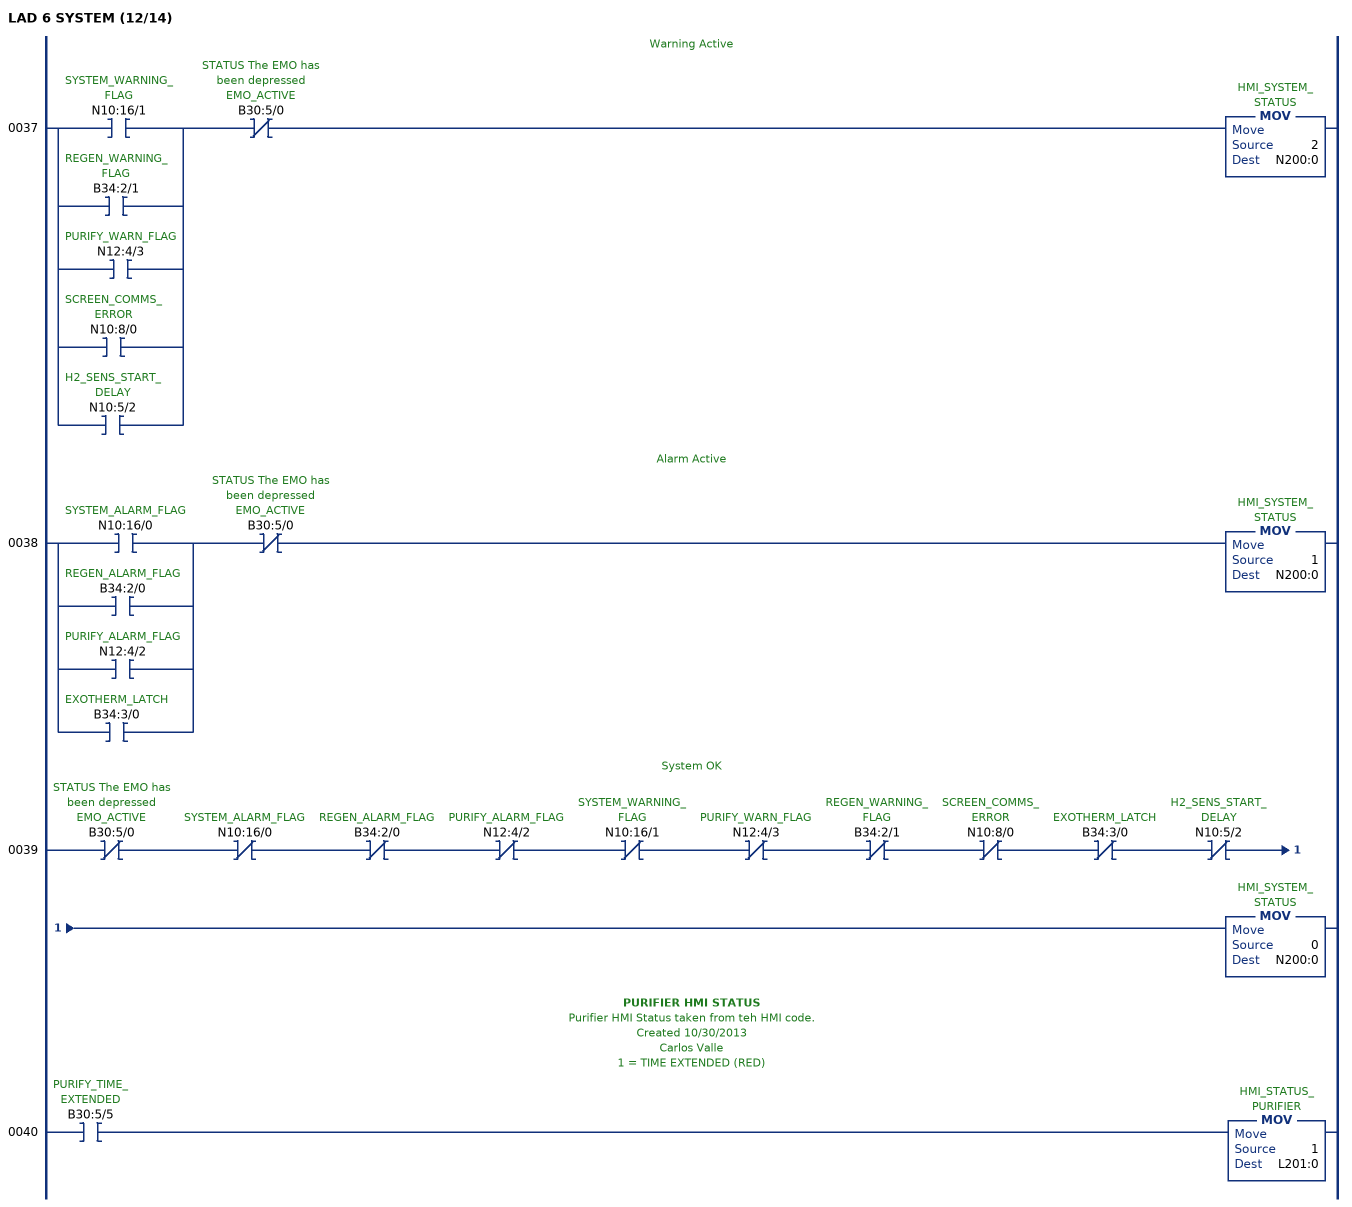
% Rung: 37 %
% Warning Active %
SOR BST XIC N10:16/1 NXB XIC B34:2/1 NXB XIC N12:4/3 NXB XIC N10:8/0 NXB XIC N10:5/2 BND XIO B30:5/0 MOV 2 N200:0 EOR
%   N10:16/1  SYSTEM_WARNING_FLAG %
%   B34:2/1  REGEN_WARNING_FLAG %
%   N12:4/3  PURIFY_WARN_FLAG %
%   N10:8/0  SCREEN_COMMS_ERROR %
%   N10:5/2  H2_SENS_START_DELAY %
%   B30:5/0  EMO_ACTIVE  "STATUS The EMO has been depressed" %
%   N200:0  HMI_SYSTEM_STATUS %
% Rung: 38 %
% Alarm Active %
SOR BST XIC N10:16/0 NXB XIC B34:2/0 NXB XIC N12:4/2 NXB XIC B34:3/0 BND XIO B30:5/0 MOV 1 N200:0 EOR
%   N10:16/0  SYSTEM_ALARM_FLAG %
%   B34:2/0  REGEN_ALARM_FLAG %
%   N12:4/2  PURIFY_ALARM_FLAG %
%   B34:3/0  EXOTHERM_LATCH %
%   B30:5/0  EMO_ACTIVE  "STATUS The EMO has been depressed" %
%   N200:0  HMI_SYSTEM_STATUS %
% Rung: 39 %
% System OK %
SOR XIO B30:5/0 XIO N10:16/0 XIO B34:2/0 XIO N12:4/2 XIO N10:16/1 XIO N12:4/3 XIO B34:2/1 XIO N10:8/0 XIO B34:3/0 XIO N10:5/2 MOV 0 N200:0 EOR
%   B30:5/0  EMO_ACTIVE  "STATUS The EMO has been depressed" %
%   N10:16/0  SYSTEM_ALARM_FLAG %
%   B34:2/0  REGEN_ALARM_FLAG %
%   N12:4/2  PURIFY_ALARM_FLAG %
%   N10:16/1  SYSTEM_WARNING_FLAG %
%   N12:4/3  PURIFY_WARN_FLAG %
%   B34:2/1  REGEN_WARNING_FLAG %
%   N10:8/0  SCREEN_COMMS_ERROR %
%   B34:3/0  EXOTHERM_LATCH %
%   N10:5/2  H2_SENS_START_DELAY %
%   N200:0  HMI_SYSTEM_STATUS %
% Rung: 40 %
% TITLE: PURIFIER HMI STATUS %
% Purifier HMI Status taken from teh HMI code.
% Created 10/30/2013
% Carlos Valle
% 1 = TIME EXTENDED (RED) %
SOR XIC B30:5/5 MOV 1 L201:0 EOR
%   B30:5/5  PURIFY_TIME_EXTENDED %
%   L201:0  HMI_STATUS_PURIFIER %

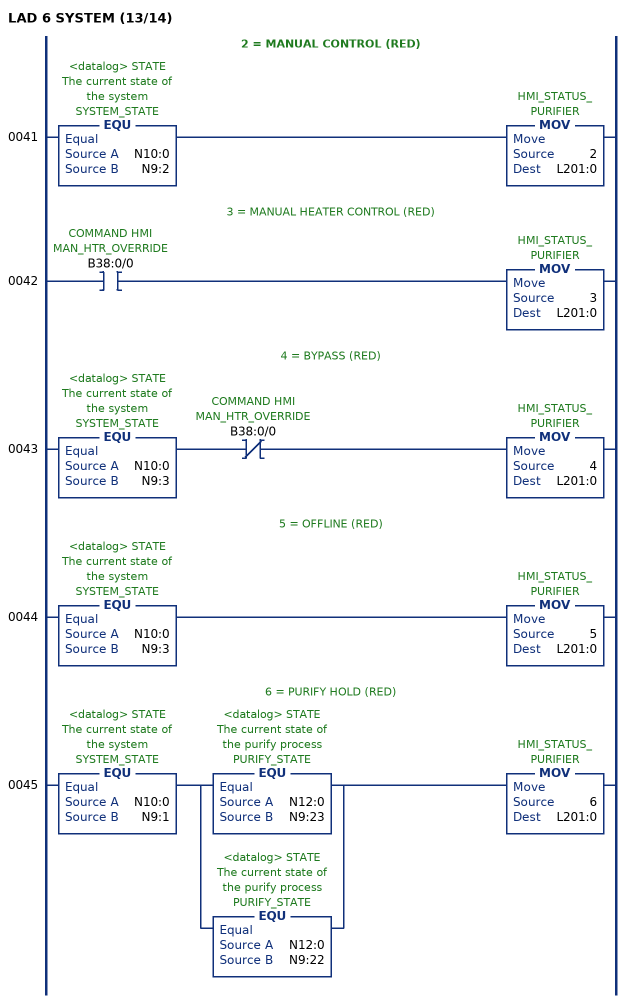
% Rung: 41 %
% TITLE: 2 = MANUAL CONTROL (RED) %
SOR EQU N10:0 N9:2 MOV 2 L201:0 EOR
%   N10:0  SYSTEM_STATE  "<datalog> STATE The current state of the system" %
%   N9:2  SYSTEM_MANUAL  "STATE System Manual" %
%   L201:0  HMI_STATUS_PURIFIER %
% Rung: 42 %
% 3 = MANUAL HEATER CONTROL (RED) %
SOR XIC B38:0/0 MOV 3 L201:0 EOR
%   B38:0/0  MAN_HTR_OVERRIDE  "COMMAND HMI" %
%   L201:0  HMI_STATUS_PURIFIER %
% Rung: 43 %
% 4 = BYPASS (RED) %
SOR EQU N10:0 N9:3 XIO B38:0/0 MOV 4 L201:0 EOR
%   N10:0  SYSTEM_STATE  "<datalog> STATE The current state of the system" %
%   N9:3  SYSTEM_ALARM  "STATE System Alarm" %
%   B38:0/0  MAN_HTR_OVERRIDE  "COMMAND HMI" %
%   L201:0  HMI_STATUS_PURIFIER %
% Rung: 44 %
% 5 = OFFLINE (RED) %
SOR EQU N10:0 N9:3 MOV 5 L201:0 EOR
%   N10:0  SYSTEM_STATE  "<datalog> STATE The current state of the system" %
%   N9:3  SYSTEM_ALARM  "STATE System Alarm" %
%   L201:0  HMI_STATUS_PURIFIER %
% Rung: 45 %
% 6 = PURIFY HOLD (RED) %
SOR EQU N10:0 N9:1 BST EQU N12:0 N9:23 NXB EQU N12:0 N9:22 BND MOV 6 L201:0 EOR
%   N10:0  SYSTEM_STATE  "<datalog> STATE The current state of the system" %
%   N9:1  SYSTEM_PROCESS  "STATE System Process" %
%   N12:0  PURIFY_STATE  "<datalog> STATE The current state of the purify process" %
%   N9:23  PURIFY_MANUAL_HOLD  "STATE Purify Manual Hold" %
%   N9:22  PURIFY_HOLD  "STATE Purify Hold" %
%   L201:0  HMI_STATUS_PURIFIER %

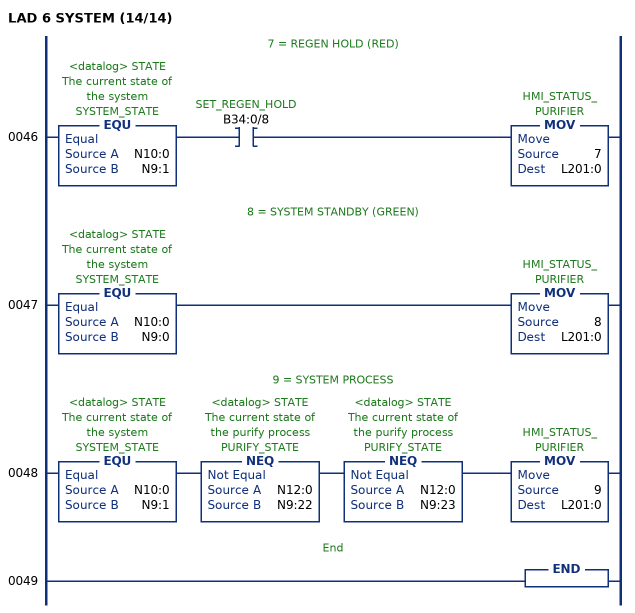
% Rung: 46 %
% 7 = REGEN HOLD (RED) %
SOR EQU N10:0 N9:1 XIC B34:0/8 MOV 7 L201:0 EOR
%   N10:0  SYSTEM_STATE  "<datalog> STATE The current state of the system" %
%   N9:1  SYSTEM_PROCESS  "STATE System Process" %
%   B34:0/8  SET_REGEN_HOLD %
%   L201:0  HMI_STATUS_PURIFIER %
% Rung: 47 %
% 8 = SYSTEM STANDBY (GREEN) %
SOR EQU N10:0 N9:0 MOV 8 L201:0 EOR
%   N10:0  SYSTEM_STATE  "<datalog> STATE The current state of the system" %
%   N9:0  SYSTEM_STANDBY  "STATE System Standby" %
%   L201:0  HMI_STATUS_PURIFIER %
% Rung: 48 %
% 9 = SYSTEM PROCESS %
SOR EQU N10:0 N9:1 NEQ N12:0 N9:22 NEQ N12:0 N9:23 MOV 9 L201:0 EOR
%   N10:0  SYSTEM_STATE  "<datalog> STATE The current state of the system" %
%   N9:1  SYSTEM_PROCESS  "STATE System Process" %
%   N12:0  PURIFY_STATE  "<datalog> STATE The current state of the purify process" %
%   N9:22  PURIFY_HOLD  "STATE Purify Hold" %
%   N9:23  PURIFY_MANUAL_HOLD  "STATE Purify Manual Hold" %
%   L201:0  HMI_STATUS_PURIFIER %
% Rung: 49 %
% End %
SOR END EOR

LADDER 7 "PROCESSING"    % Runs the processing control %
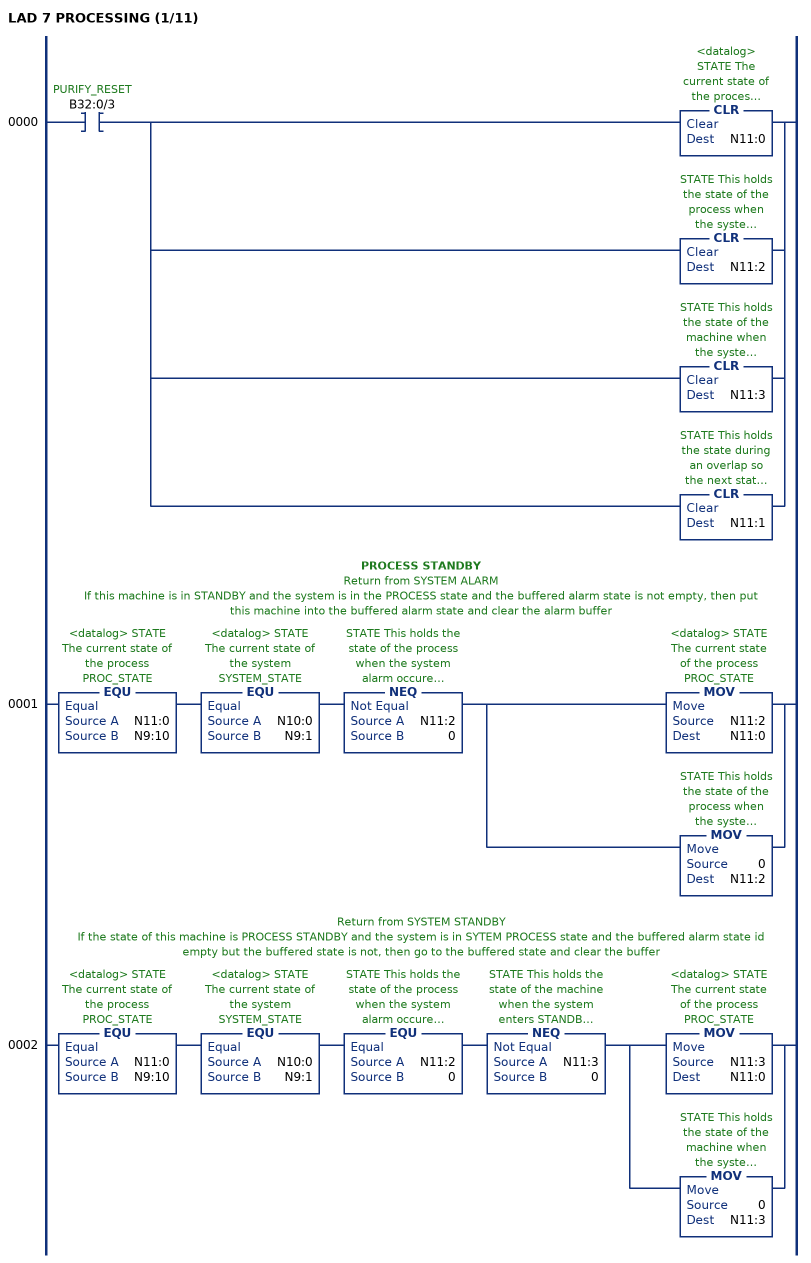
% Rung: 0 %
SOR XIC B32:0/3 BST CLR N11:0 NXB CLR N11:2 NXB CLR N11:3 NXB CLR N11:1 BND EOR
%   B32:0/3  PURIFY_RESET %
%   N11:0  PROC_STATE  "<datalog> STATE The current state of the process" %
%   N11:2  PROC_ALARM_BUFFER  "STATE This holds the state of the process when the system alarm occured" %
%   N11:3  PROC_STANDBY_BUFFER  "STATE This holds the state of the machine when the system enters STANDBY state" %
%   N11:1  PROC_OVERLAP_BUFFER  "STATE This holds the state during an overlap so the next state can be determined" %
% Rung: 1 %
% TITLE: PROCESS STANDBY %
% Return from SYSTEM ALARM
% If this machine is in STANDBY and the system is in the PROCESS state and the buffered alarm state is not empty, then put this machine into the buffered alarm state and clear the alarm buffer %
SOR EQU N11:0 N9:10 EQU N10:0 N9:1 NEQ N11:2 0 BST MOV N11:2 N11:0 NXB MOV 0 N11:2 BND EOR
%   N11:0  PROC_STATE  "<datalog> STATE The current state of the process" %
%   N9:10  PROCESS_STANDBY  "STATE Process Standby" %
%   N10:0  SYSTEM_STATE  "<datalog> STATE The current state of the system" %
%   N9:1  SYSTEM_PROCESS  "STATE System Process" %
%   N11:2  PROC_ALARM_BUFFER  "STATE This holds the state of the process when the system alarm occured" %
% Rung: 2 %
% Return from SYSTEM STANDBY
% If the state of this machine is PROCESS STANDBY and the system is in SYTEM PROCESS state and the buffered alarm state id empty but the buffered state is not, then go to the buffered state and clear the buffer %
SOR EQU N11:0 N9:10 EQU N10:0 N9:1 EQU N11:2 0 NEQ N11:3 0 BST MOV N11:3 N11:0 NXB MOV 0 N11:3 BND EOR
%   N11:0  PROC_STATE  "<datalog> STATE The current state of the process" %
%   N9:10  PROCESS_STANDBY  "STATE Process Standby" %
%   N10:0  SYSTEM_STATE  "<datalog> STATE The current state of the system" %
%   N9:1  SYSTEM_PROCESS  "STATE System Process" %
%   N11:2  PROC_ALARM_BUFFER  "STATE This holds the state of the process when the system alarm occured" %
%   N11:3  PROC_STANDBY_BUFFER  "STATE This holds the state of the machine when the system enters STANDBY state" %

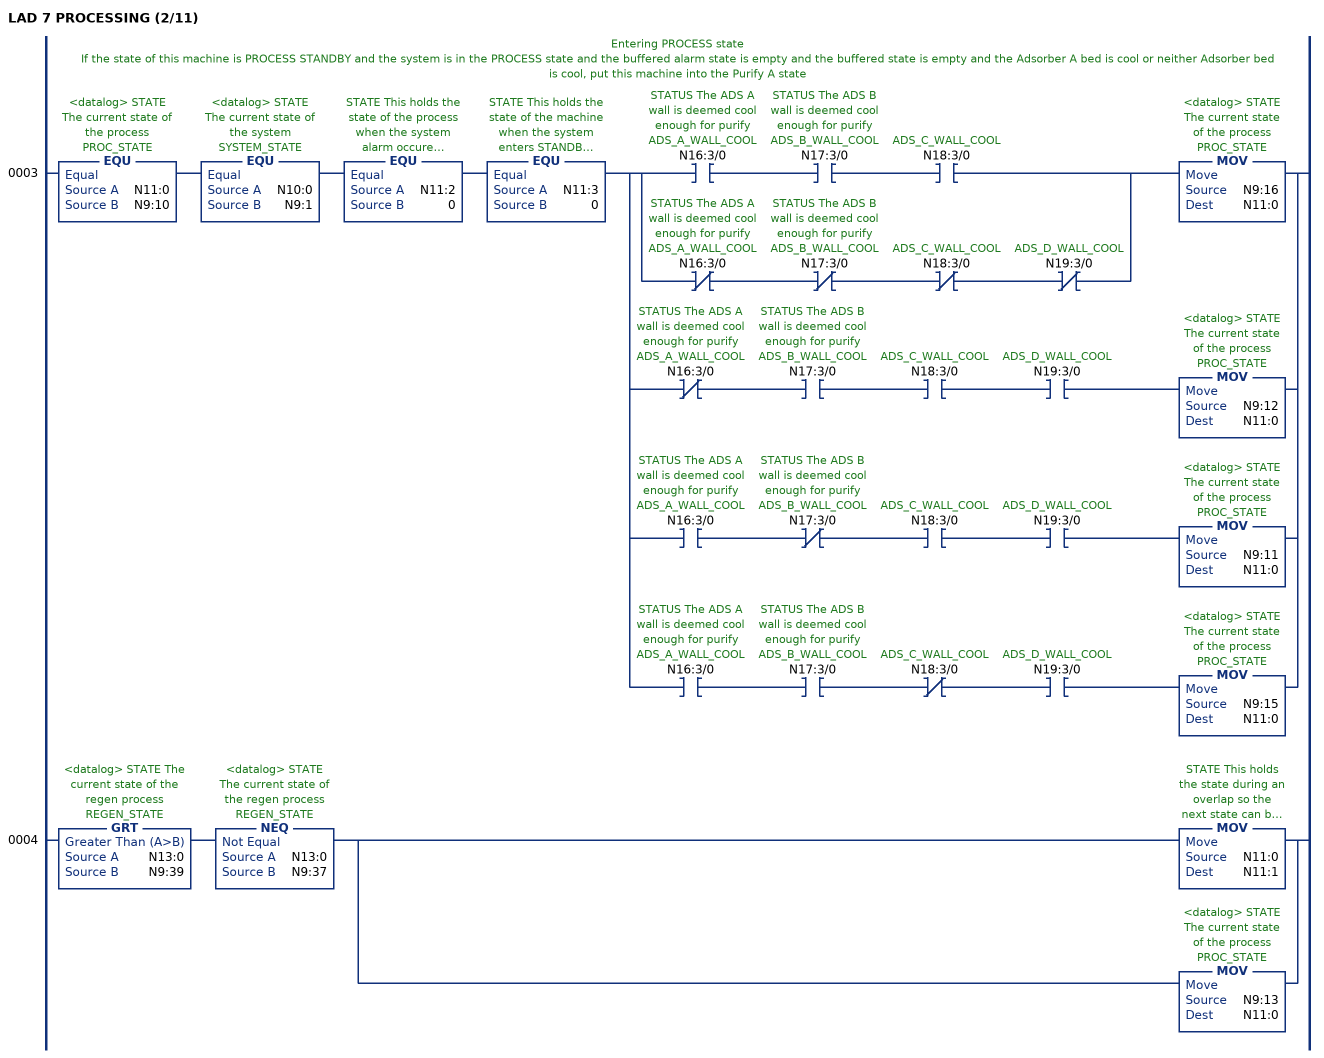
% Rung: 3 %
% Entering PROCESS state
% If the state of this machine is PROCESS STANDBY and the system is in the PROCESS state and the buffered alarm state is empty and the buffered state is empty and the Adsorber A bed is cool or neither Adsorber bed is cool, put this machine into the Purify A state %
SOR EQU N11:0 N9:10 EQU N10:0 N9:1 EQU N11:2 0 EQU N11:3 0 BST BST XIC N16:3/0 XIC N17:3/0 XIC N18:3/0 NXB XIO N16:3/0 XIO N17:3/0 XIO N18:3/0 XIO N19:3/0 BND MOV N9:16 N11:0 NXB XIO N16:3/0 XIC N17:3/0 XIC N18:3/0 XIC N19:3/0 MOV N9:12 N11:0 NXB XIC N16:3/0 XIO N17:3/0 XIC N18:3/0 XIC N19:3/0 MOV N9:11 N11:0 NXB XIC N16:3/0 XIC N17:3/0 XIO N18:3/0 XIC N19:3/0 MOV N9:15 N11:0 BND EOR
%   N11:0  PROC_STATE  "<datalog> STATE The current state of the process" %
%   N9:10  PROCESS_STANDBY  "STATE Process Standby" %
%   N10:0  SYSTEM_STATE  "<datalog> STATE The current state of the system" %
%   N9:1  SYSTEM_PROCESS  "STATE System Process" %
%   N11:2  PROC_ALARM_BUFFER  "STATE This holds the state of the process when the system alarm occured" %
%   N11:3  PROC_STANDBY_BUFFER  "STATE This holds the state of the machine when the system enters STANDBY state" %
%   N16:3/0  ADS_A_WALL_COOL  "STATUS The ADS A wall is deemed cool enough for purify" %
%   N17:3/0  ADS_B_WALL_COOL  "STATUS The ADS B wall is deemed cool enough for purify" %
%   N18:3/0  ADS_C_WALL_COOL %
%   N19:3/0  ADS_D_WALL_COOL %
%   N9:16  PROC_REGEN_D  "STATE Process Regen D" %
%   N9:12  PROC_REGEN_A  "STATE Process Regen A" %
%   N9:11  PROC_REGEN_B  "STATE Process Regen B" %
%   N9:15  PROC_REGEN_C  "STATE Process Regen C" %
% Rung: 4 %
SOR GRT N13:0 N9:39 NEQ N13:0 N9:37 BST MOV N11:0 N11:1 NXB MOV N9:13 N11:0 BND EOR
%   N13:0  REGEN_STATE  "<datalog> STATE The current state of the regen process" %
%   N9:39  REGEN_EQUALIZE  "STATE Regen Equalize" %
%   N9:37  REGEN_ALARM  "STATE Regen Alarm" %
%   N11:0  PROC_STATE  "<datalog> STATE The current state of the process" %
%   N11:1  PROC_OVERLAP_BUFFER  "STATE This holds the state during an overlap so the next state can be determined" %
%   N9:13  PROC_OVERLAP  "STATE Process Purify Overlap" %

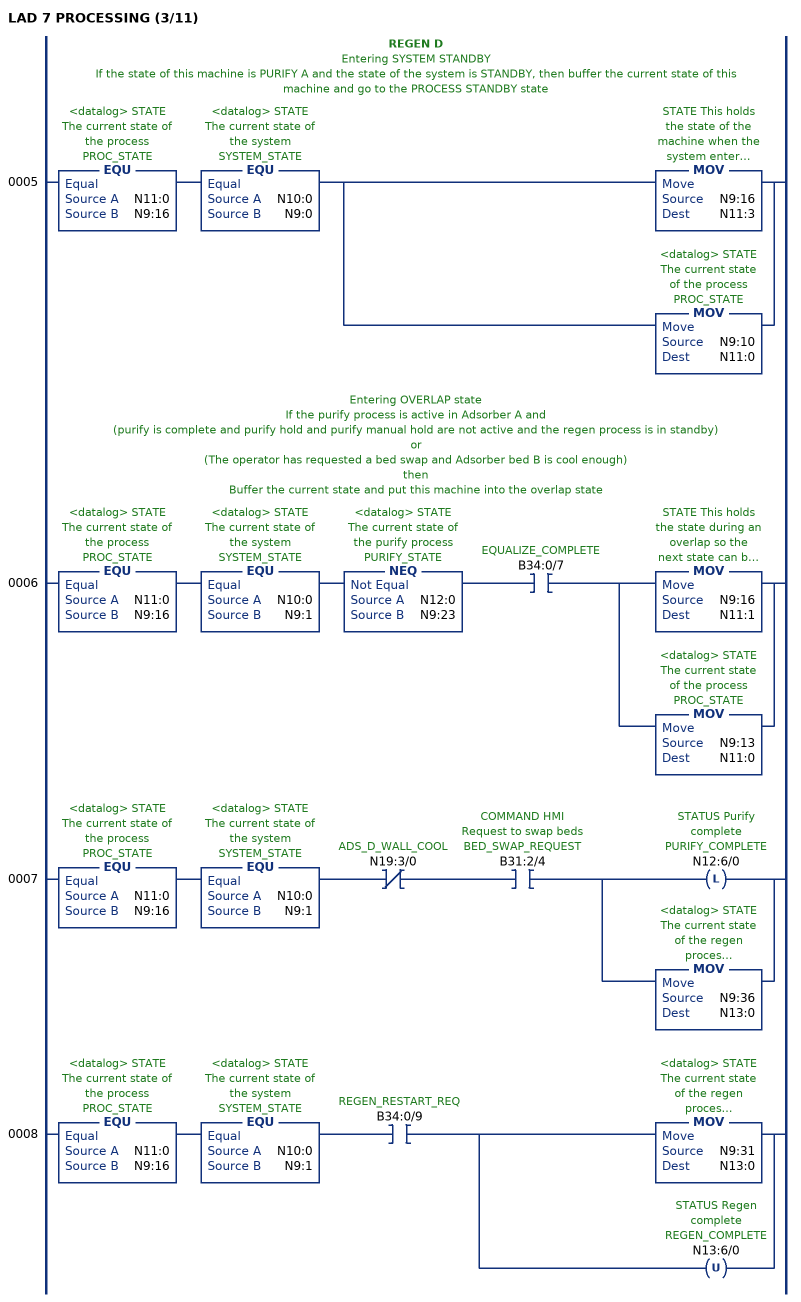
% Rung: 5 %
% TITLE: REGEN D %
% Entering SYSTEM STANDBY
% If the state of this machine is PURIFY A and the state of the system is STANDBY, then buffer the current state of this machine and go to the PROCESS STANDBY state %
SOR EQU N11:0 N9:16 EQU N10:0 N9:0 BST MOV N9:16 N11:3 NXB MOV N9:10 N11:0 BND EOR
%   N11:0  PROC_STATE  "<datalog> STATE The current state of the process" %
%   N9:16  PROC_REGEN_D  "STATE Process Regen D" %
%   N10:0  SYSTEM_STATE  "<datalog> STATE The current state of the system" %
%   N9:0  SYSTEM_STANDBY  "STATE System Standby" %
%   N11:3  PROC_STANDBY_BUFFER  "STATE This holds the state of the machine when the system enters STANDBY state" %
%   N9:10  PROCESS_STANDBY  "STATE Process Standby" %
% Rung: 6 %
% Entering OVERLAP state
% If the purify process is active in Adsorber A and
% (purify is complete and purify hold and purify manual hold are not active and the regen process is in standby)
% or
% (The operator has requested a bed swap and Adsorber bed B is cool enough)
% then
% Buffer the current state and put this machine into the overlap state %
SOR EQU N11:0 N9:16 EQU N10:0 N9:1 NEQ N12:0 N9:23 XIC B34:0/7 BST MOV N9:16 N11:1 NXB MOV N9:13 N11:0 BND EOR
%   N11:0  PROC_STATE  "<datalog> STATE The current state of the process" %
%   N9:16  PROC_REGEN_D  "STATE Process Regen D" %
%   N10:0  SYSTEM_STATE  "<datalog> STATE The current state of the system" %
%   N9:1  SYSTEM_PROCESS  "STATE System Process" %
%   N12:0  PURIFY_STATE  "<datalog> STATE The current state of the purify process" %
%   N9:23  PURIFY_MANUAL_HOLD  "STATE Purify Manual Hold" %
%   B34:0/7  EQUALIZE_COMPLETE %
%   N11:1  PROC_OVERLAP_BUFFER  "STATE This holds the state during an overlap so the next state can be determined" %
%   N9:13  PROC_OVERLAP  "STATE Process Purify Overlap" %
% Rung: 7 %
SOR EQU N11:0 N9:16 EQU N10:0 N9:1 XIO N19:3/0 XIC B31:2/4 BST OTL N12:6/0 NXB MOV N9:36 N13:0 BND EOR
%   N11:0  PROC_STATE  "<datalog> STATE The current state of the process" %
%   N9:16  PROC_REGEN_D  "STATE Process Regen D" %
%   N10:0  SYSTEM_STATE  "<datalog> STATE The current state of the system" %
%   N9:1  SYSTEM_PROCESS  "STATE System Process" %
%   N19:3/0  ADS_D_WALL_COOL %
%   B31:2/4  BED_SWAP_REQUEST  "COMMAND HMI Request to swap beds" %
%   N12:6/0  PURIFY_COMPLETE  "STATUS Purify complete" %
%   N9:36  REGEN_COOL  "STATE Regen Cool" %
%   N13:0  REGEN_STATE  "<datalog> STATE The current state of the regen process" %
% Rung: 8 %
SOR EQU N11:0 N9:16 EQU N10:0 N9:1 XIC B34:0/9 BST MOV N9:31 N13:0 NXB OTU N13:6/0 BND EOR
%   N11:0  PROC_STATE  "<datalog> STATE The current state of the process" %
%   N9:16  PROC_REGEN_D  "STATE Process Regen D" %
%   N10:0  SYSTEM_STATE  "<datalog> STATE The current state of the system" %
%   N9:1  SYSTEM_PROCESS  "STATE System Process" %
%   B34:0/9  REGEN_RESTART_REQ %
%   N9:31  REGEN_DELAY  "STATE Regen Delay" %
%   N13:0  REGEN_STATE  "<datalog> STATE The current state of the regen process" %
%   N13:6/0  REGEN_COMPLETE  "STATUS Regen complete" %

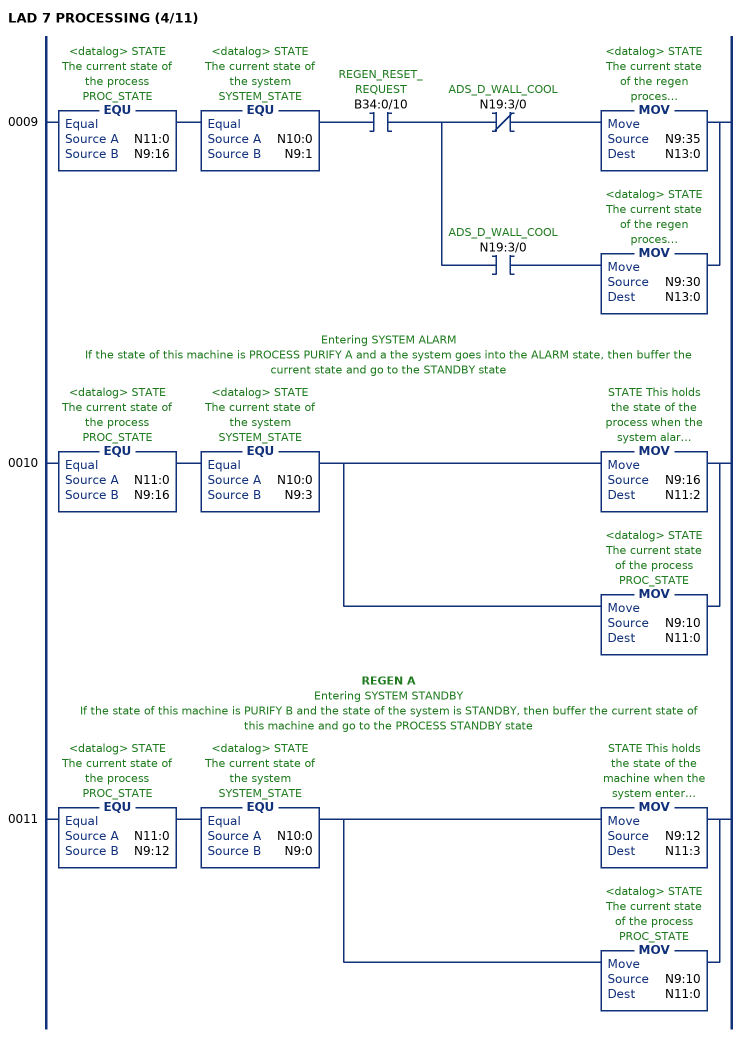
% Rung: 9 %
SOR EQU N11:0 N9:16 EQU N10:0 N9:1 XIC B34:0/10 BST XIO N19:3/0 MOV N9:35 N13:0 NXB XIC N19:3/0 MOV N9:30 N13:0 BND EOR
%   N11:0  PROC_STATE  "<datalog> STATE The current state of the process" %
%   N9:16  PROC_REGEN_D  "STATE Process Regen D" %
%   N10:0  SYSTEM_STATE  "<datalog> STATE The current state of the system" %
%   N9:1  SYSTEM_PROCESS  "STATE System Process" %
%   B34:0/10  REGEN_RESET_REQUEST %
%   N19:3/0  ADS_D_WALL_COOL %
%   N9:35  REGEN_COOL_WALL  "STATE Regen Cool wall" %
%   N13:0  REGEN_STATE  "<datalog> STATE The current state of the regen process" %
%   N9:30  REGEN_STANDBY  "STATE Regen Standby" %
% Rung: 10 %
% Entering SYSTEM ALARM
% If the state of this machine is PROCESS PURIFY A and a the system goes into the ALARM state, then buffer the current state and go to the STANDBY state %
SOR EQU N11:0 N9:16 EQU N10:0 N9:3 BST MOV N9:16 N11:2 NXB MOV N9:10 N11:0 BND EOR
%   N11:0  PROC_STATE  "<datalog> STATE The current state of the process" %
%   N9:16  PROC_REGEN_D  "STATE Process Regen D" %
%   N10:0  SYSTEM_STATE  "<datalog> STATE The current state of the system" %
%   N9:3  SYSTEM_ALARM  "STATE System Alarm" %
%   N11:2  PROC_ALARM_BUFFER  "STATE This holds the state of the process when the system alarm occured" %
%   N9:10  PROCESS_STANDBY  "STATE Process Standby" %
% Rung: 11 %
% TITLE: REGEN A %
% Entering SYSTEM STANDBY
% If the state of this machine is PURIFY B and the state of the system is STANDBY, then buffer the current state of this machine and go to the PROCESS STANDBY state %
SOR EQU N11:0 N9:12 EQU N10:0 N9:0 BST MOV N9:12 N11:3 NXB MOV N9:10 N11:0 BND EOR
%   N11:0  PROC_STATE  "<datalog> STATE The current state of the process" %
%   N9:12  PROC_REGEN_A  "STATE Process Regen A" %
%   N10:0  SYSTEM_STATE  "<datalog> STATE The current state of the system" %
%   N9:0  SYSTEM_STANDBY  "STATE System Standby" %
%   N11:3  PROC_STANDBY_BUFFER  "STATE This holds the state of the machine when the system enters STANDBY state" %
%   N9:10  PROCESS_STANDBY  "STATE Process Standby" %

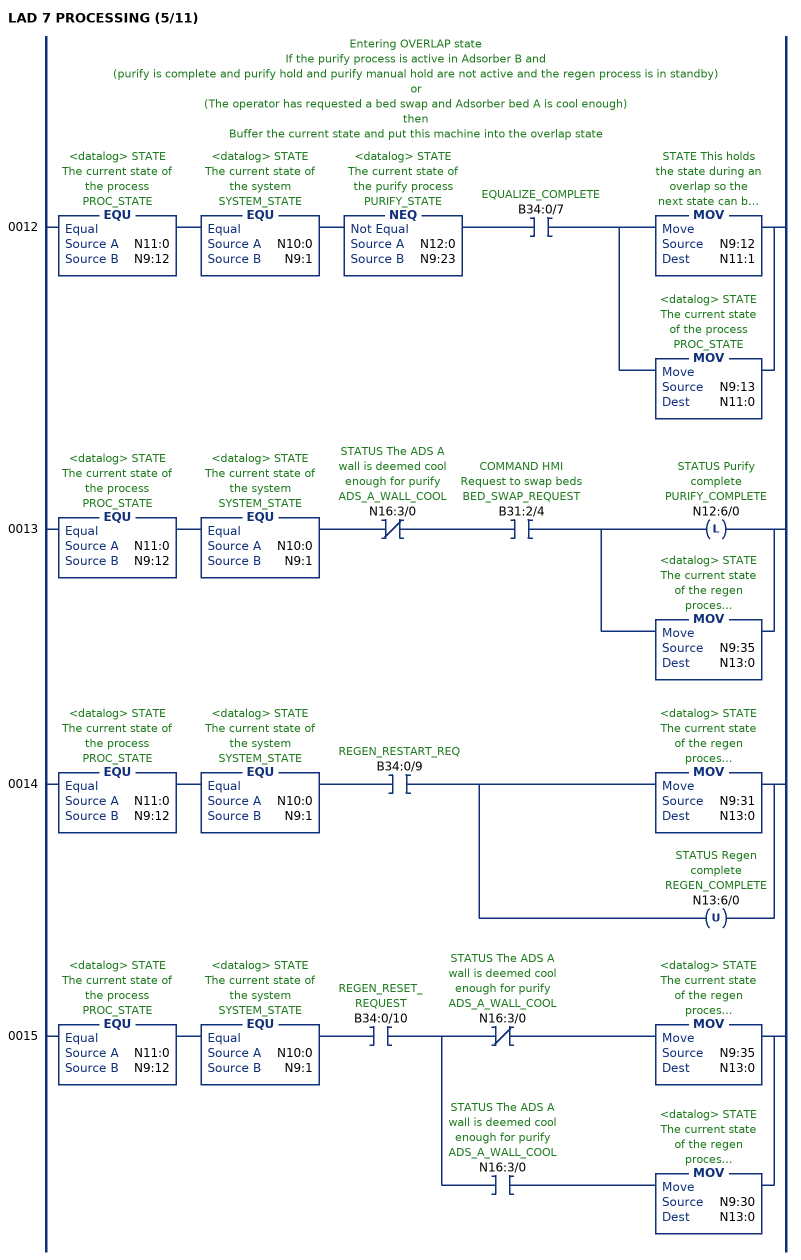
% Rung: 12 %
% Entering OVERLAP state
% If the purify process is active in Adsorber B and
% (purify is complete and purify hold and purify manual hold are not active and the regen process is in standby)
% or
% (The operator has requested a bed swap and Adsorber bed A is cool enough)
% then
% Buffer the current state and put this machine into the overlap state %
SOR EQU N11:0 N9:12 EQU N10:0 N9:1 NEQ N12:0 N9:23 XIC B34:0/7 BST MOV N9:12 N11:1 NXB MOV N9:13 N11:0 BND EOR
%   N11:0  PROC_STATE  "<datalog> STATE The current state of the process" %
%   N9:12  PROC_REGEN_A  "STATE Process Regen A" %
%   N10:0  SYSTEM_STATE  "<datalog> STATE The current state of the system" %
%   N9:1  SYSTEM_PROCESS  "STATE System Process" %
%   N12:0  PURIFY_STATE  "<datalog> STATE The current state of the purify process" %
%   N9:23  PURIFY_MANUAL_HOLD  "STATE Purify Manual Hold" %
%   B34:0/7  EQUALIZE_COMPLETE %
%   N11:1  PROC_OVERLAP_BUFFER  "STATE This holds the state during an overlap so the next state can be determined" %
%   N9:13  PROC_OVERLAP  "STATE Process Purify Overlap" %
% Rung: 13 %
SOR EQU N11:0 N9:12 EQU N10:0 N9:1 XIO N16:3/0 XIC B31:2/4 BST OTL N12:6/0 NXB MOV N9:35 N13:0 BND EOR
%   N11:0  PROC_STATE  "<datalog> STATE The current state of the process" %
%   N9:12  PROC_REGEN_A  "STATE Process Regen A" %
%   N10:0  SYSTEM_STATE  "<datalog> STATE The current state of the system" %
%   N9:1  SYSTEM_PROCESS  "STATE System Process" %
%   N16:3/0  ADS_A_WALL_COOL  "STATUS The ADS A wall is deemed cool enough for purify" %
%   B31:2/4  BED_SWAP_REQUEST  "COMMAND HMI Request to swap beds" %
%   N12:6/0  PURIFY_COMPLETE  "STATUS Purify complete" %
%   N9:35  REGEN_COOL_WALL  "STATE Regen Cool wall" %
%   N13:0  REGEN_STATE  "<datalog> STATE The current state of the regen process" %
% Rung: 14 %
SOR EQU N11:0 N9:12 EQU N10:0 N9:1 XIC B34:0/9 BST MOV N9:31 N13:0 NXB OTU N13:6/0 BND EOR
%   N11:0  PROC_STATE  "<datalog> STATE The current state of the process" %
%   N9:12  PROC_REGEN_A  "STATE Process Regen A" %
%   N10:0  SYSTEM_STATE  "<datalog> STATE The current state of the system" %
%   N9:1  SYSTEM_PROCESS  "STATE System Process" %
%   B34:0/9  REGEN_RESTART_REQ %
%   N9:31  REGEN_DELAY  "STATE Regen Delay" %
%   N13:0  REGEN_STATE  "<datalog> STATE The current state of the regen process" %
%   N13:6/0  REGEN_COMPLETE  "STATUS Regen complete" %
% Rung: 15 %
SOR EQU N11:0 N9:12 EQU N10:0 N9:1 XIC B34:0/10 BST XIO N16:3/0 MOV N9:35 N13:0 NXB XIC N16:3/0 MOV N9:30 N13:0 BND EOR
%   N11:0  PROC_STATE  "<datalog> STATE The current state of the process" %
%   N9:12  PROC_REGEN_A  "STATE Process Regen A" %
%   N10:0  SYSTEM_STATE  "<datalog> STATE The current state of the system" %
%   N9:1  SYSTEM_PROCESS  "STATE System Process" %
%   B34:0/10  REGEN_RESET_REQUEST %
%   N16:3/0  ADS_A_WALL_COOL  "STATUS The ADS A wall is deemed cool enough for purify" %
%   N9:35  REGEN_COOL_WALL  "STATE Regen Cool wall" %
%   N13:0  REGEN_STATE  "<datalog> STATE The current state of the regen process" %
%   N9:30  REGEN_STANDBY  "STATE Regen Standby" %

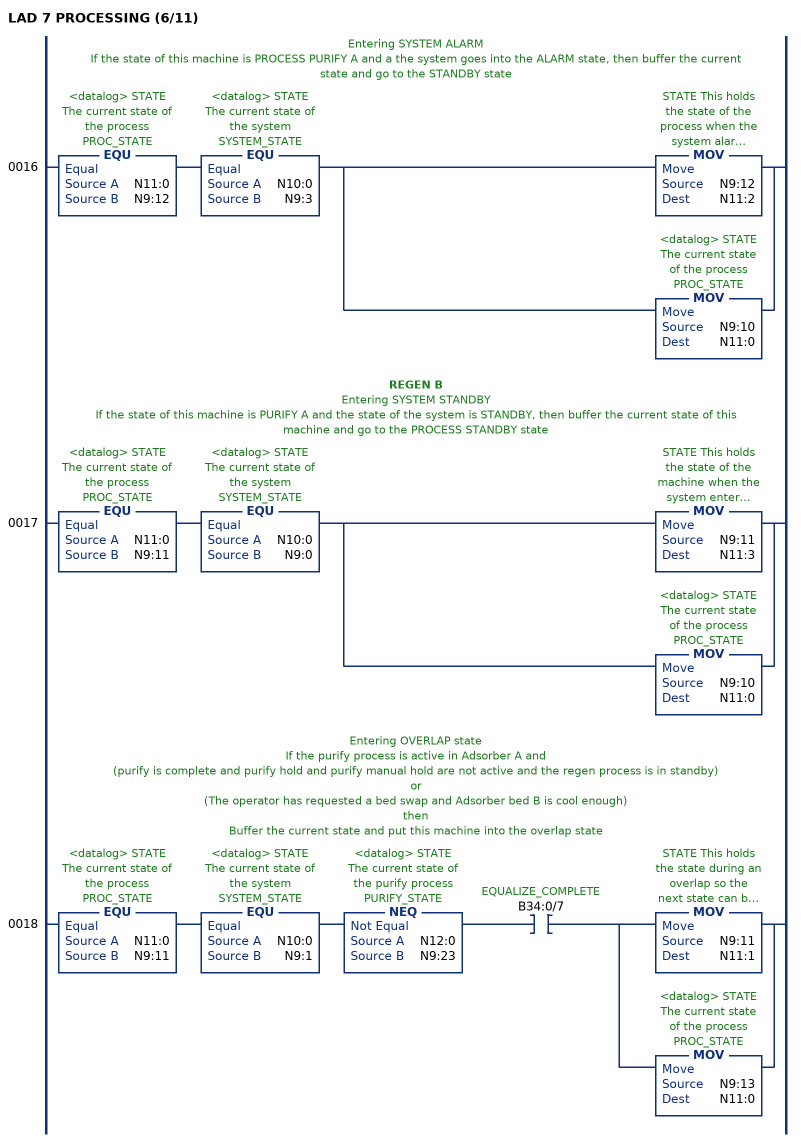
% Rung: 16 %
% Entering SYSTEM ALARM
% If the state of this machine is PROCESS PURIFY A and a the system goes into the ALARM state, then buffer the current state and go to the STANDBY state %
SOR EQU N11:0 N9:12 EQU N10:0 N9:3 BST MOV N9:12 N11:2 NXB MOV N9:10 N11:0 BND EOR
%   N11:0  PROC_STATE  "<datalog> STATE The current state of the process" %
%   N9:12  PROC_REGEN_A  "STATE Process Regen A" %
%   N10:0  SYSTEM_STATE  "<datalog> STATE The current state of the system" %
%   N9:3  SYSTEM_ALARM  "STATE System Alarm" %
%   N11:2  PROC_ALARM_BUFFER  "STATE This holds the state of the process when the system alarm occured" %
%   N9:10  PROCESS_STANDBY  "STATE Process Standby" %
% Rung: 17 %
% TITLE: REGEN B %
% Entering SYSTEM STANDBY
% If the state of this machine is PURIFY A and the state of the system is STANDBY, then buffer the current state of this machine and go to the PROCESS STANDBY state %
SOR EQU N11:0 N9:11 EQU N10:0 N9:0 BST MOV N9:11 N11:3 NXB MOV N9:10 N11:0 BND EOR
%   N11:0  PROC_STATE  "<datalog> STATE The current state of the process" %
%   N9:11  PROC_REGEN_B  "STATE Process Regen B" %
%   N10:0  SYSTEM_STATE  "<datalog> STATE The current state of the system" %
%   N9:0  SYSTEM_STANDBY  "STATE System Standby" %
%   N11:3  PROC_STANDBY_BUFFER  "STATE This holds the state of the machine when the system enters STANDBY state" %
%   N9:10  PROCESS_STANDBY  "STATE Process Standby" %
% Rung: 18 %
% Entering OVERLAP state
% If the purify process is active in Adsorber A and
% (purify is complete and purify hold and purify manual hold are not active and the regen process is in standby)
% or
% (The operator has requested a bed swap and Adsorber bed B is cool enough)
% then
% Buffer the current state and put this machine into the overlap state %
SOR EQU N11:0 N9:11 EQU N10:0 N9:1 NEQ N12:0 N9:23 XIC B34:0/7 BST MOV N9:11 N11:1 NXB MOV N9:13 N11:0 BND EOR
%   N11:0  PROC_STATE  "<datalog> STATE The current state of the process" %
%   N9:11  PROC_REGEN_B  "STATE Process Regen B" %
%   N10:0  SYSTEM_STATE  "<datalog> STATE The current state of the system" %
%   N9:1  SYSTEM_PROCESS  "STATE System Process" %
%   N12:0  PURIFY_STATE  "<datalog> STATE The current state of the purify process" %
%   N9:23  PURIFY_MANUAL_HOLD  "STATE Purify Manual Hold" %
%   B34:0/7  EQUALIZE_COMPLETE %
%   N11:1  PROC_OVERLAP_BUFFER  "STATE This holds the state during an overlap so the next state can be determined" %
%   N9:13  PROC_OVERLAP  "STATE Process Purify Overlap" %

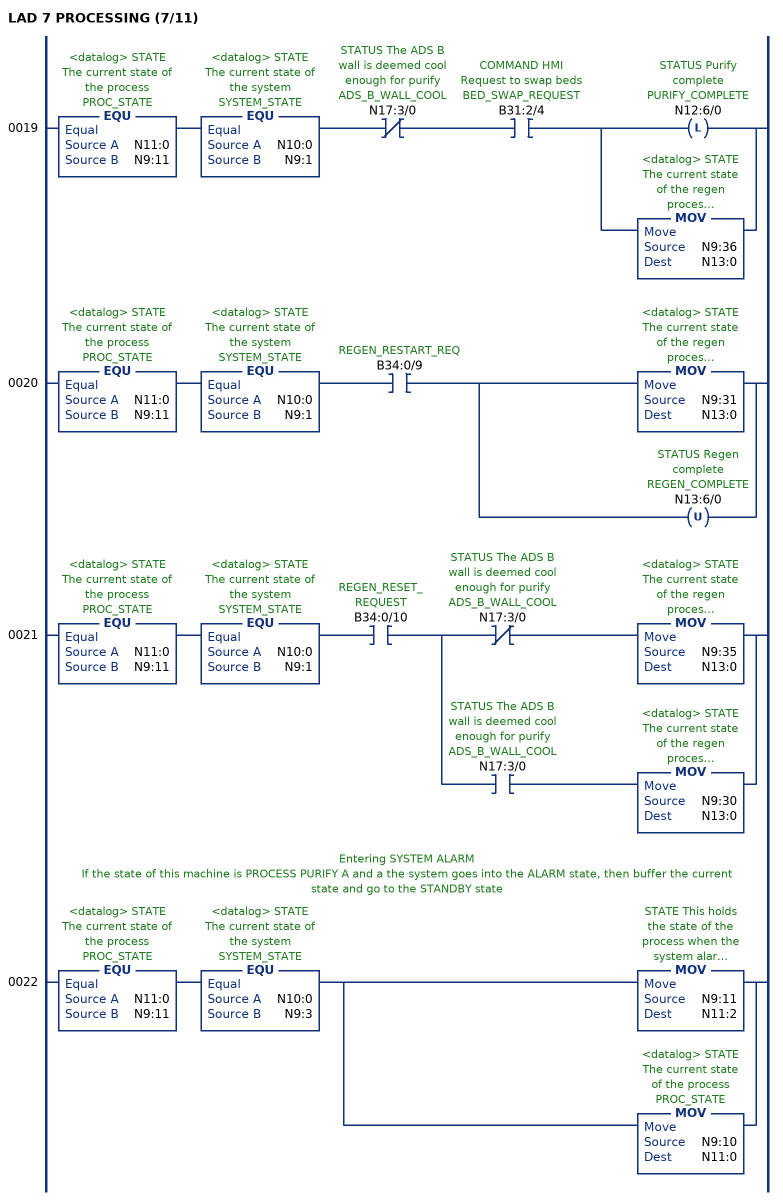
% Rung: 19 %
SOR EQU N11:0 N9:11 EQU N10:0 N9:1 XIO N17:3/0 XIC B31:2/4 BST OTL N12:6/0 NXB MOV N9:36 N13:0 BND EOR
%   N11:0  PROC_STATE  "<datalog> STATE The current state of the process" %
%   N9:11  PROC_REGEN_B  "STATE Process Regen B" %
%   N10:0  SYSTEM_STATE  "<datalog> STATE The current state of the system" %
%   N9:1  SYSTEM_PROCESS  "STATE System Process" %
%   N17:3/0  ADS_B_WALL_COOL  "STATUS The ADS B wall is deemed cool enough for purify" %
%   B31:2/4  BED_SWAP_REQUEST  "COMMAND HMI Request to swap beds" %
%   N12:6/0  PURIFY_COMPLETE  "STATUS Purify complete" %
%   N9:36  REGEN_COOL  "STATE Regen Cool" %
%   N13:0  REGEN_STATE  "<datalog> STATE The current state of the regen process" %
% Rung: 20 %
SOR EQU N11:0 N9:11 EQU N10:0 N9:1 XIC B34:0/9 BST MOV N9:31 N13:0 NXB OTU N13:6/0 BND EOR
%   N11:0  PROC_STATE  "<datalog> STATE The current state of the process" %
%   N9:11  PROC_REGEN_B  "STATE Process Regen B" %
%   N10:0  SYSTEM_STATE  "<datalog> STATE The current state of the system" %
%   N9:1  SYSTEM_PROCESS  "STATE System Process" %
%   B34:0/9  REGEN_RESTART_REQ %
%   N9:31  REGEN_DELAY  "STATE Regen Delay" %
%   N13:0  REGEN_STATE  "<datalog> STATE The current state of the regen process" %
%   N13:6/0  REGEN_COMPLETE  "STATUS Regen complete" %
% Rung: 21 %
SOR EQU N11:0 N9:11 EQU N10:0 N9:1 XIC B34:0/10 BST XIO N17:3/0 MOV N9:35 N13:0 NXB XIC N17:3/0 MOV N9:30 N13:0 BND EOR
%   N11:0  PROC_STATE  "<datalog> STATE The current state of the process" %
%   N9:11  PROC_REGEN_B  "STATE Process Regen B" %
%   N10:0  SYSTEM_STATE  "<datalog> STATE The current state of the system" %
%   N9:1  SYSTEM_PROCESS  "STATE System Process" %
%   B34:0/10  REGEN_RESET_REQUEST %
%   N17:3/0  ADS_B_WALL_COOL  "STATUS The ADS B wall is deemed cool enough for purify" %
%   N9:35  REGEN_COOL_WALL  "STATE Regen Cool wall" %
%   N13:0  REGEN_STATE  "<datalog> STATE The current state of the regen process" %
%   N9:30  REGEN_STANDBY  "STATE Regen Standby" %
% Rung: 22 %
% Entering SYSTEM ALARM
% If the state of this machine is PROCESS PURIFY A and a the system goes into the ALARM state, then buffer the current state and go to the STANDBY state %
SOR EQU N11:0 N9:11 EQU N10:0 N9:3 BST MOV N9:11 N11:2 NXB MOV N9:10 N11:0 BND EOR
%   N11:0  PROC_STATE  "<datalog> STATE The current state of the process" %
%   N9:11  PROC_REGEN_B  "STATE Process Regen B" %
%   N10:0  SYSTEM_STATE  "<datalog> STATE The current state of the system" %
%   N9:3  SYSTEM_ALARM  "STATE System Alarm" %
%   N11:2  PROC_ALARM_BUFFER  "STATE This holds the state of the process when the system alarm occured" %
%   N9:10  PROCESS_STANDBY  "STATE Process Standby" %

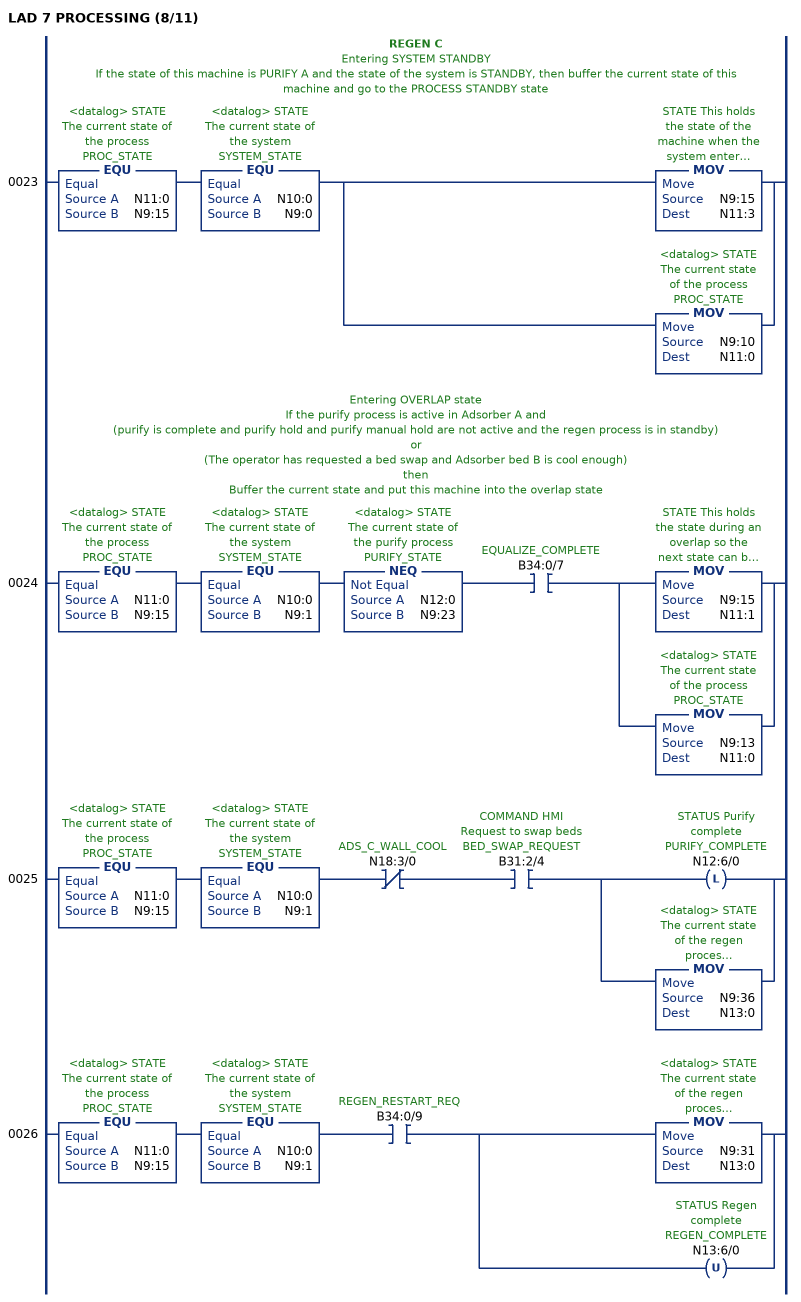
% Rung: 23 %
% TITLE: REGEN C %
% Entering SYSTEM STANDBY
% If the state of this machine is PURIFY A and the state of the system is STANDBY, then buffer the current state of this machine and go to the PROCESS STANDBY state %
SOR EQU N11:0 N9:15 EQU N10:0 N9:0 BST MOV N9:15 N11:3 NXB MOV N9:10 N11:0 BND EOR
%   N11:0  PROC_STATE  "<datalog> STATE The current state of the process" %
%   N9:15  PROC_REGEN_C  "STATE Process Regen C" %
%   N10:0  SYSTEM_STATE  "<datalog> STATE The current state of the system" %
%   N9:0  SYSTEM_STANDBY  "STATE System Standby" %
%   N11:3  PROC_STANDBY_BUFFER  "STATE This holds the state of the machine when the system enters STANDBY state" %
%   N9:10  PROCESS_STANDBY  "STATE Process Standby" %
% Rung: 24 %
% Entering OVERLAP state
% If the purify process is active in Adsorber A and
% (purify is complete and purify hold and purify manual hold are not active and the regen process is in standby)
% or
% (The operator has requested a bed swap and Adsorber bed B is cool enough)
% then
% Buffer the current state and put this machine into the overlap state %
SOR EQU N11:0 N9:15 EQU N10:0 N9:1 NEQ N12:0 N9:23 XIC B34:0/7 BST MOV N9:15 N11:1 NXB MOV N9:13 N11:0 BND EOR
%   N11:0  PROC_STATE  "<datalog> STATE The current state of the process" %
%   N9:15  PROC_REGEN_C  "STATE Process Regen C" %
%   N10:0  SYSTEM_STATE  "<datalog> STATE The current state of the system" %
%   N9:1  SYSTEM_PROCESS  "STATE System Process" %
%   N12:0  PURIFY_STATE  "<datalog> STATE The current state of the purify process" %
%   N9:23  PURIFY_MANUAL_HOLD  "STATE Purify Manual Hold" %
%   B34:0/7  EQUALIZE_COMPLETE %
%   N11:1  PROC_OVERLAP_BUFFER  "STATE This holds the state during an overlap so the next state can be determined" %
%   N9:13  PROC_OVERLAP  "STATE Process Purify Overlap" %
% Rung: 25 %
SOR EQU N11:0 N9:15 EQU N10:0 N9:1 XIO N18:3/0 XIC B31:2/4 BST OTL N12:6/0 NXB MOV N9:36 N13:0 BND EOR
%   N11:0  PROC_STATE  "<datalog> STATE The current state of the process" %
%   N9:15  PROC_REGEN_C  "STATE Process Regen C" %
%   N10:0  SYSTEM_STATE  "<datalog> STATE The current state of the system" %
%   N9:1  SYSTEM_PROCESS  "STATE System Process" %
%   N18:3/0  ADS_C_WALL_COOL %
%   B31:2/4  BED_SWAP_REQUEST  "COMMAND HMI Request to swap beds" %
%   N12:6/0  PURIFY_COMPLETE  "STATUS Purify complete" %
%   N9:36  REGEN_COOL  "STATE Regen Cool" %
%   N13:0  REGEN_STATE  "<datalog> STATE The current state of the regen process" %
% Rung: 26 %
SOR EQU N11:0 N9:15 EQU N10:0 N9:1 XIC B34:0/9 BST MOV N9:31 N13:0 NXB OTU N13:6/0 BND EOR
%   N11:0  PROC_STATE  "<datalog> STATE The current state of the process" %
%   N9:15  PROC_REGEN_C  "STATE Process Regen C" %
%   N10:0  SYSTEM_STATE  "<datalog> STATE The current state of the system" %
%   N9:1  SYSTEM_PROCESS  "STATE System Process" %
%   B34:0/9  REGEN_RESTART_REQ %
%   N9:31  REGEN_DELAY  "STATE Regen Delay" %
%   N13:0  REGEN_STATE  "<datalog> STATE The current state of the regen process" %
%   N13:6/0  REGEN_COMPLETE  "STATUS Regen complete" %

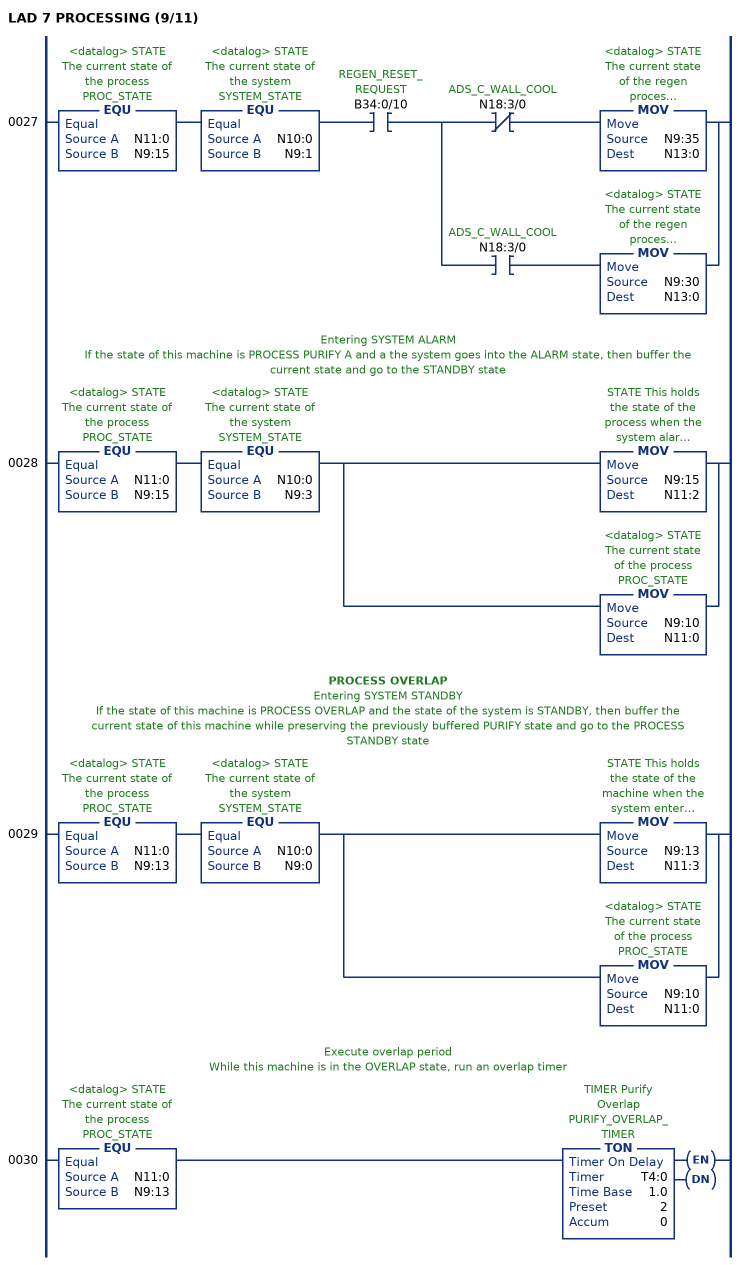
% Rung: 27 %
SOR EQU N11:0 N9:15 EQU N10:0 N9:1 XIC B34:0/10 BST XIO N18:3/0 MOV N9:35 N13:0 NXB XIC N18:3/0 MOV N9:30 N13:0 BND EOR
%   N11:0  PROC_STATE  "<datalog> STATE The current state of the process" %
%   N9:15  PROC_REGEN_C  "STATE Process Regen C" %
%   N10:0  SYSTEM_STATE  "<datalog> STATE The current state of the system" %
%   N9:1  SYSTEM_PROCESS  "STATE System Process" %
%   B34:0/10  REGEN_RESET_REQUEST %
%   N18:3/0  ADS_C_WALL_COOL %
%   N9:35  REGEN_COOL_WALL  "STATE Regen Cool wall" %
%   N13:0  REGEN_STATE  "<datalog> STATE The current state of the regen process" %
%   N9:30  REGEN_STANDBY  "STATE Regen Standby" %
% Rung: 28 %
% Entering SYSTEM ALARM
% If the state of this machine is PROCESS PURIFY A and a the system goes into the ALARM state, then buffer the current state and go to the STANDBY state %
SOR EQU N11:0 N9:15 EQU N10:0 N9:3 BST MOV N9:15 N11:2 NXB MOV N9:10 N11:0 BND EOR
%   N11:0  PROC_STATE  "<datalog> STATE The current state of the process" %
%   N9:15  PROC_REGEN_C  "STATE Process Regen C" %
%   N10:0  SYSTEM_STATE  "<datalog> STATE The current state of the system" %
%   N9:3  SYSTEM_ALARM  "STATE System Alarm" %
%   N11:2  PROC_ALARM_BUFFER  "STATE This holds the state of the process when the system alarm occured" %
%   N9:10  PROCESS_STANDBY  "STATE Process Standby" %
% Rung: 29 %
% TITLE: PROCESS OVERLAP %
% Entering SYSTEM STANDBY
% If the state of this machine is PROCESS OVERLAP and the state of the system is STANDBY, then buffer the current state of this machine while preserving the previously buffered PURIFY state and go to the PROCESS STANDBY state %
SOR EQU N11:0 N9:13 EQU N10:0 N9:0 BST MOV N9:13 N11:3 NXB MOV N9:10 N11:0 BND EOR
%   N11:0  PROC_STATE  "<datalog> STATE The current state of the process" %
%   N9:13  PROC_OVERLAP  "STATE Process Purify Overlap" %
%   N10:0  SYSTEM_STATE  "<datalog> STATE The current state of the system" %
%   N9:0  SYSTEM_STANDBY  "STATE System Standby" %
%   N11:3  PROC_STANDBY_BUFFER  "STATE This holds the state of the machine when the system enters STANDBY state" %
%   N9:10  PROCESS_STANDBY  "STATE Process Standby" %
% Rung: 30 %
% Execute overlap period
% While this machine is in the OVERLAP state, run an overlap timer %
SOR EQU N11:0 N9:13 TON T4:0 1.0 2 0 EOR
%   N11:0  PROC_STATE  "<datalog> STATE The current state of the process" %
%   N9:13  PROC_OVERLAP  "STATE Process Purify Overlap" %
%   T4:0  PURIFY_OVERLAP_TIMER  "TIMER Purify Overlap" %

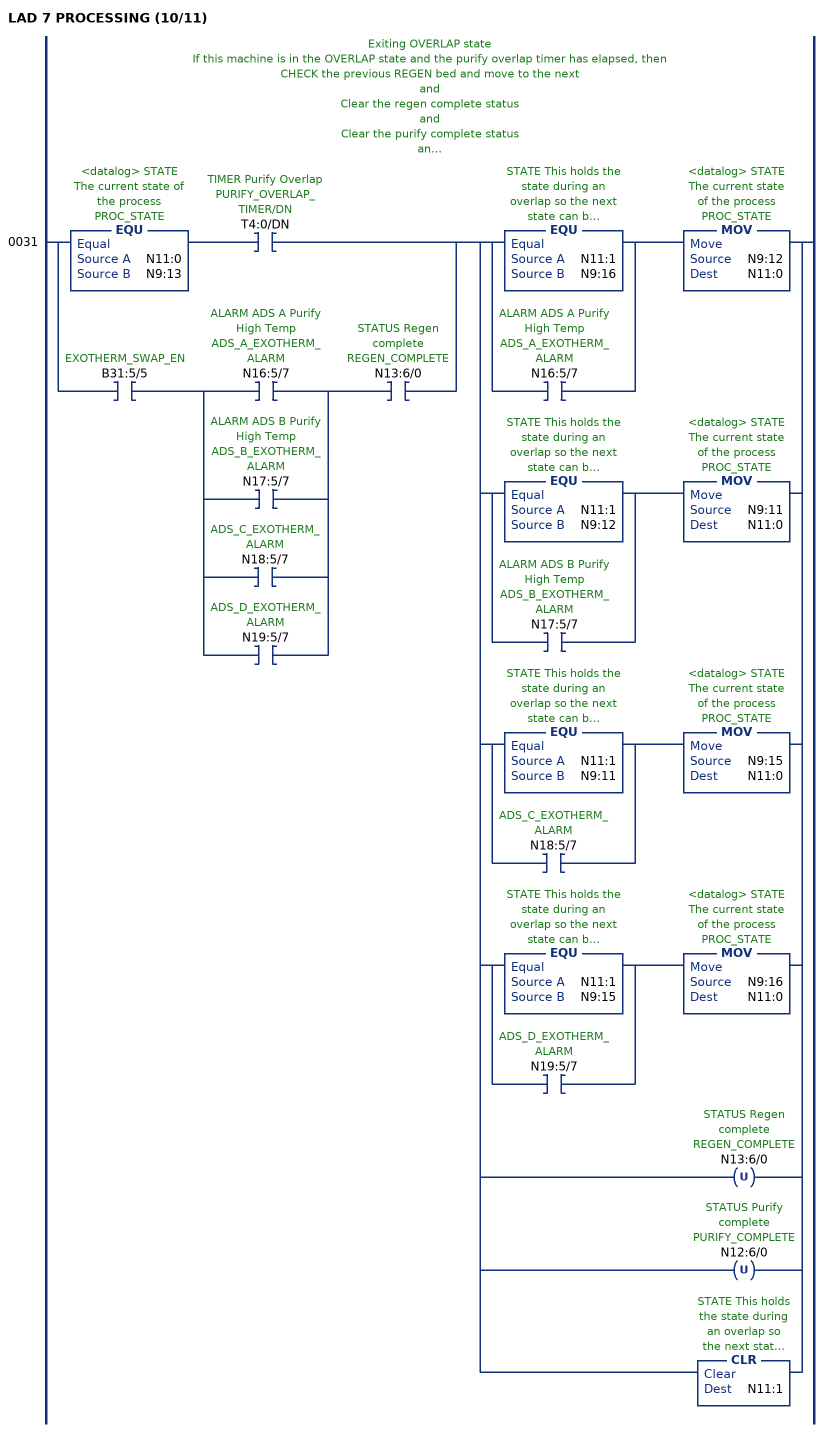
% Rung: 31 %
% Exiting OVERLAP state
% If this machine is in the OVERLAP state and the purify overlap timer has elapsed, then
% CHECK the previous REGEN bed and move to the next
% and
% Clear the regen complete status
% and
% Clear the purify complete status
% and
% clear the process buffer %
SOR BST EQU N11:0 N9:13 XIC T4:0/DN NXB XIC B31:5/5 BST XIC N16:5/7 NXB XIC N17:5/7 NXB XIC N18:5/7 NXB XIC N19:5/7 BND XIC N13:6/0 BND BST BST EQU N11:1 N9:16 NXB XIC N16:5/7 BND MOV N9:12 N11:0 NXB BST EQU N11:1 N9:12 NXB XIC N17:5/7 BND MOV N9:11 N11:0 NXB BST EQU N11:1 N9:11 NXB XIC N18:5/7 BND MOV N9:15 N11:0 NXB BST EQU N11:1 N9:15 NXB XIC N19:5/7 BND MOV N9:16 N11:0 NXB OTU N13:6/0 NXB OTU N12:6/0 NXB CLR N11:1 BND EOR
%   N11:0  PROC_STATE  "<datalog> STATE The current state of the process" %
%   N9:13  PROC_OVERLAP  "STATE Process Purify Overlap" %
%   T4:0  PURIFY_OVERLAP_TIMER  "TIMER Purify Overlap" %
%   B31:5/5  EXOTHERM_SWAP_EN %
%   N16:5/7  ADS_A_EXOTHERM_ALARM  "ALARM ADS A Purify High Temp" %
%   N17:5/7  ADS_B_EXOTHERM_ALARM  "ALARM ADS B Purify High Temp" %
%   N18:5/7  ADS_C_EXOTHERM_ALARM %
%   N19:5/7  ADS_D_EXOTHERM_ALARM %
%   N13:6/0  REGEN_COMPLETE  "STATUS Regen complete" %
%   N11:1  PROC_OVERLAP_BUFFER  "STATE This holds the state during an overlap so the next state can be determined" %
%   N9:16  PROC_REGEN_D  "STATE Process Regen D" %
%   N9:12  PROC_REGEN_A  "STATE Process Regen A" %
%   N9:11  PROC_REGEN_B  "STATE Process Regen B" %
%   N9:15  PROC_REGEN_C  "STATE Process Regen C" %
%   N12:6/0  PURIFY_COMPLETE  "STATUS Purify complete" %

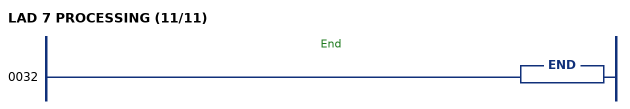
% Rung: 32 %
% End %
SOR END EOR

LADDER 8 "MANUAL_CTL"    % Runs the manual valve control %
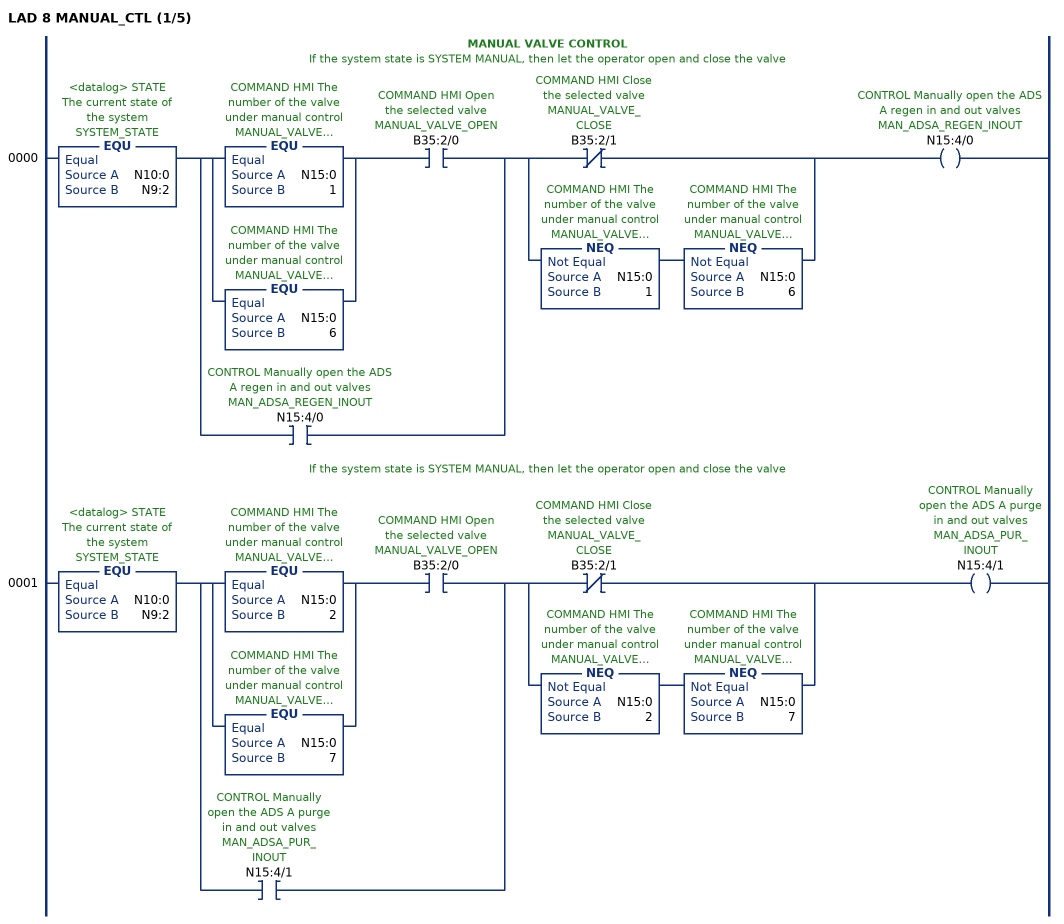
% Rung: 0 %
% TITLE: MANUAL VALVE CONTROL %
% If the system state is SYSTEM MANUAL, then let the operator open and close the valve %
SOR EQU N10:0 N9:2 BST BST EQU N15:0 1 NXB EQU N15:0 6 BND XIC B35:2/0 NXB XIC N15:4/0 BND BST XIO B35:2/1 NXB NEQ N15:0 1 NEQ N15:0 6 BND OTE N15:4/0 EOR
%   N10:0  SYSTEM_STATE  "<datalog> STATE The current state of the system" %
%   N9:2  SYSTEM_MANUAL  "STATE System Manual" %
%   N15:0  MANUAL_VALVE_NUMBER  "COMMAND HMI The number of the valve under manual control" %
%   B35:2/0  MANUAL_VALVE_OPEN  "COMMAND HMI Open the selected valve" %
%   N15:4/0  MAN_ADSA_REGEN_INOUT  "CONTROL Manually open the ADS A regen in and out valves" %
%   B35:2/1  MANUAL_VALVE_CLOSE  "COMMAND HMI Close the selected valve" %
% Rung: 1 %
% If the system state is SYSTEM MANUAL, then let the operator open and close the valve %
SOR EQU N10:0 N9:2 BST BST EQU N15:0 2 NXB EQU N15:0 7 BND XIC B35:2/0 NXB XIC N15:4/1 BND BST XIO B35:2/1 NXB NEQ N15:0 2 NEQ N15:0 7 BND OTE N15:4/1 EOR
%   N10:0  SYSTEM_STATE  "<datalog> STATE The current state of the system" %
%   N9:2  SYSTEM_MANUAL  "STATE System Manual" %
%   N15:0  MANUAL_VALVE_NUMBER  "COMMAND HMI The number of the valve under manual control" %
%   B35:2/0  MANUAL_VALVE_OPEN  "COMMAND HMI Open the selected valve" %
%   N15:4/1  MAN_ADSA_PUR_INOUT  "CONTROL Manually open the ADS A purge in and out valves" %
%   B35:2/1  MANUAL_VALVE_CLOSE  "COMMAND HMI Close the selected valve" %

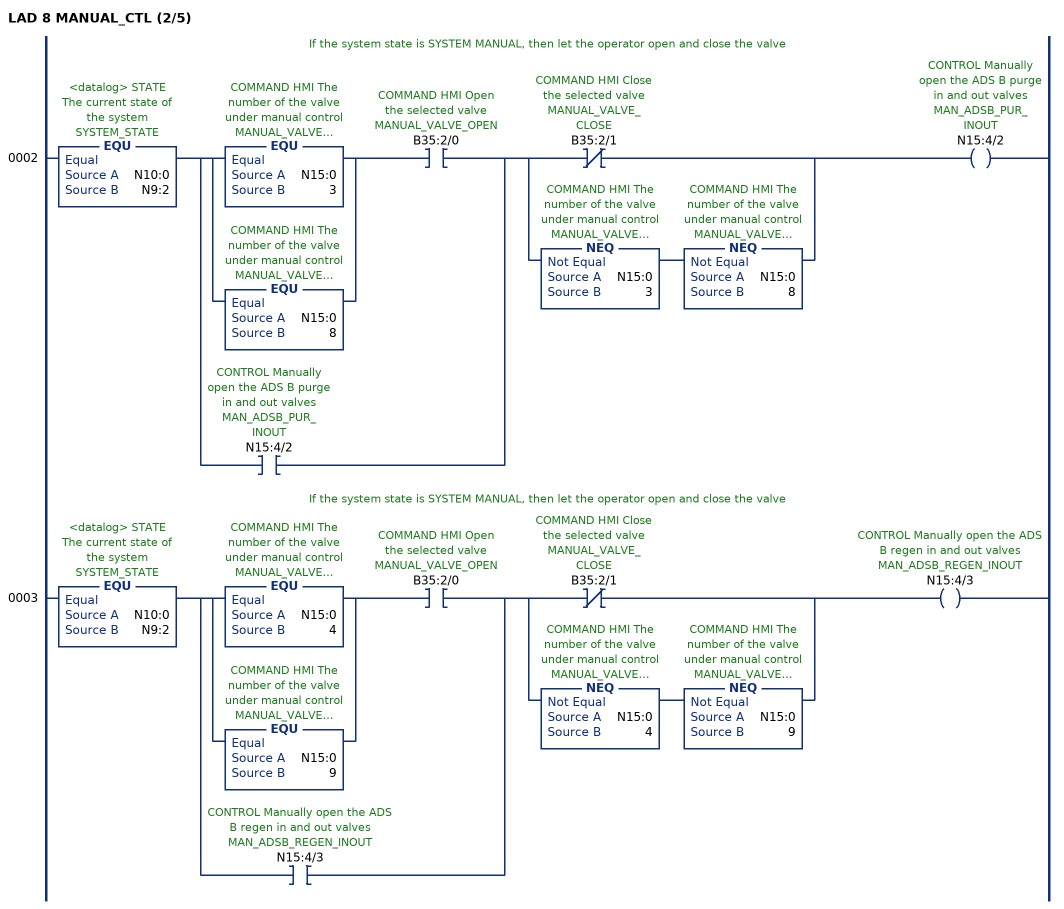
% Rung: 2 %
% If the system state is SYSTEM MANUAL, then let the operator open and close the valve %
SOR EQU N10:0 N9:2 BST BST EQU N15:0 3 NXB EQU N15:0 8 BND XIC B35:2/0 NXB XIC N15:4/2 BND BST XIO B35:2/1 NXB NEQ N15:0 3 NEQ N15:0 8 BND OTE N15:4/2 EOR
%   N10:0  SYSTEM_STATE  "<datalog> STATE The current state of the system" %
%   N9:2  SYSTEM_MANUAL  "STATE System Manual" %
%   N15:0  MANUAL_VALVE_NUMBER  "COMMAND HMI The number of the valve under manual control" %
%   B35:2/0  MANUAL_VALVE_OPEN  "COMMAND HMI Open the selected valve" %
%   N15:4/2  MAN_ADSB_PUR_INOUT  "CONTROL Manually open the ADS B purge in and out valves" %
%   B35:2/1  MANUAL_VALVE_CLOSE  "COMMAND HMI Close the selected valve" %
% Rung: 3 %
% If the system state is SYSTEM MANUAL, then let the operator open and close the valve %
SOR EQU N10:0 N9:2 BST BST EQU N15:0 4 NXB EQU N15:0 9 BND XIC B35:2/0 NXB XIC N15:4/3 BND BST XIO B35:2/1 NXB NEQ N15:0 4 NEQ N15:0 9 BND OTE N15:4/3 EOR
%   N10:0  SYSTEM_STATE  "<datalog> STATE The current state of the system" %
%   N9:2  SYSTEM_MANUAL  "STATE System Manual" %
%   N15:0  MANUAL_VALVE_NUMBER  "COMMAND HMI The number of the valve under manual control" %
%   B35:2/0  MANUAL_VALVE_OPEN  "COMMAND HMI Open the selected valve" %
%   N15:4/3  MAN_ADSB_REGEN_INOUT  "CONTROL Manually open the ADS B regen in and out valves" %
%   B35:2/1  MANUAL_VALVE_CLOSE  "COMMAND HMI Close the selected valve" %

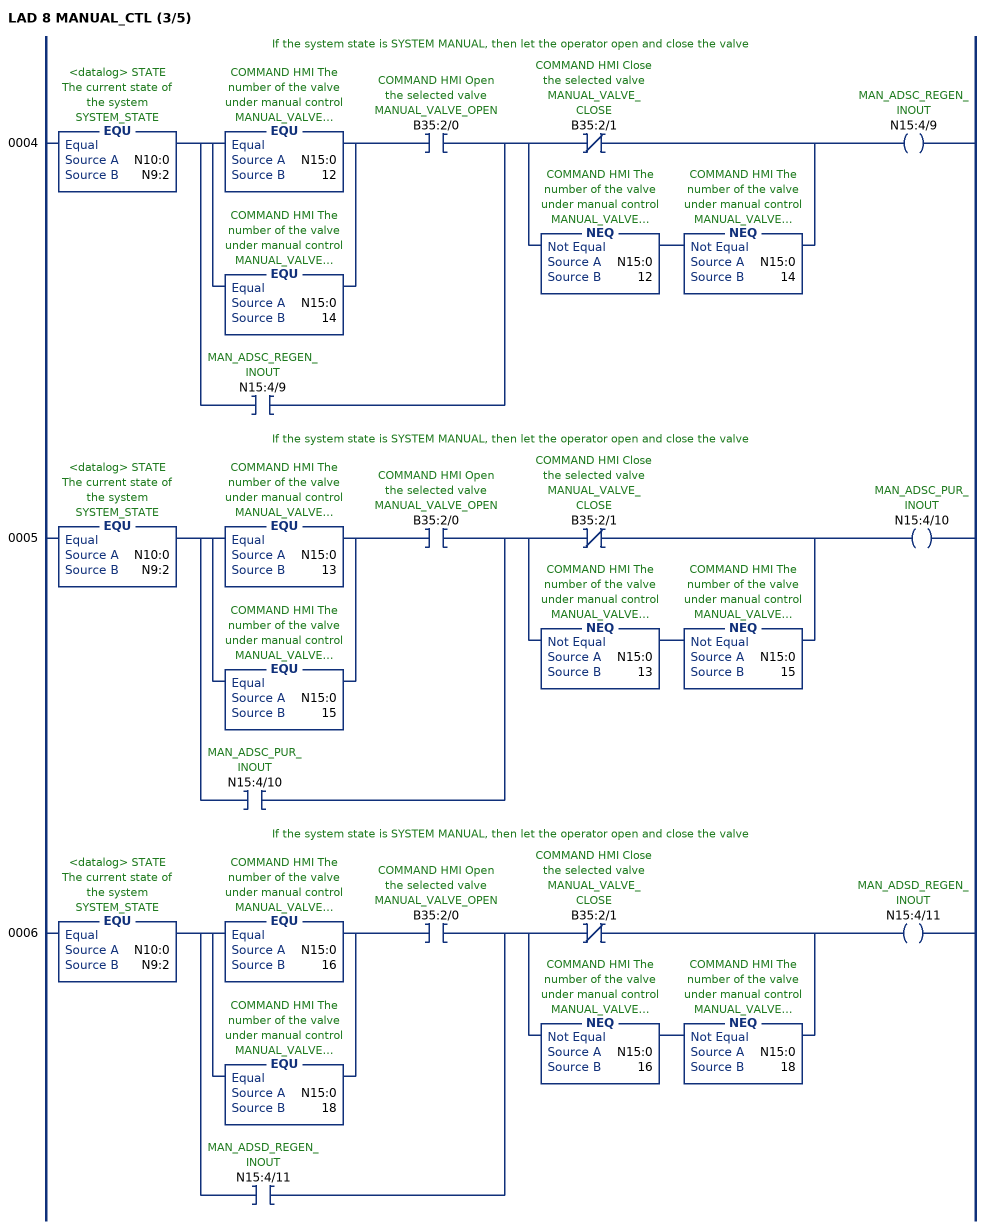
% Rung: 4 %
% If the system state is SYSTEM MANUAL, then let the operator open and close the valve %
SOR EQU N10:0 N9:2 BST BST EQU N15:0 12 NXB EQU N15:0 14 BND XIC B35:2/0 NXB XIC N15:4/9 BND BST XIO B35:2/1 NXB NEQ N15:0 12 NEQ N15:0 14 BND OTE N15:4/9 EOR
%   N10:0  SYSTEM_STATE  "<datalog> STATE The current state of the system" %
%   N9:2  SYSTEM_MANUAL  "STATE System Manual" %
%   N15:0  MANUAL_VALVE_NUMBER  "COMMAND HMI The number of the valve under manual control" %
%   B35:2/0  MANUAL_VALVE_OPEN  "COMMAND HMI Open the selected valve" %
%   N15:4/9  MAN_ADSC_REGEN_INOUT %
%   B35:2/1  MANUAL_VALVE_CLOSE  "COMMAND HMI Close the selected valve" %
% Rung: 5 %
% If the system state is SYSTEM MANUAL, then let the operator open and close the valve %
SOR EQU N10:0 N9:2 BST BST EQU N15:0 13 NXB EQU N15:0 15 BND XIC B35:2/0 NXB XIC N15:4/10 BND BST XIO B35:2/1 NXB NEQ N15:0 13 NEQ N15:0 15 BND OTE N15:4/10 EOR
%   N10:0  SYSTEM_STATE  "<datalog> STATE The current state of the system" %
%   N9:2  SYSTEM_MANUAL  "STATE System Manual" %
%   N15:0  MANUAL_VALVE_NUMBER  "COMMAND HMI The number of the valve under manual control" %
%   B35:2/0  MANUAL_VALVE_OPEN  "COMMAND HMI Open the selected valve" %
%   N15:4/10  MAN_ADSC_PUR_INOUT %
%   B35:2/1  MANUAL_VALVE_CLOSE  "COMMAND HMI Close the selected valve" %
% Rung: 6 %
% If the system state is SYSTEM MANUAL, then let the operator open and close the valve %
SOR EQU N10:0 N9:2 BST BST EQU N15:0 16 NXB EQU N15:0 18 BND XIC B35:2/0 NXB XIC N15:4/11 BND BST XIO B35:2/1 NXB NEQ N15:0 16 NEQ N15:0 18 BND OTE N15:4/11 EOR
%   N10:0  SYSTEM_STATE  "<datalog> STATE The current state of the system" %
%   N9:2  SYSTEM_MANUAL  "STATE System Manual" %
%   N15:0  MANUAL_VALVE_NUMBER  "COMMAND HMI The number of the valve under manual control" %
%   B35:2/0  MANUAL_VALVE_OPEN  "COMMAND HMI Open the selected valve" %
%   N15:4/11  MAN_ADSD_REGEN_INOUT %
%   B35:2/1  MANUAL_VALVE_CLOSE  "COMMAND HMI Close the selected valve" %

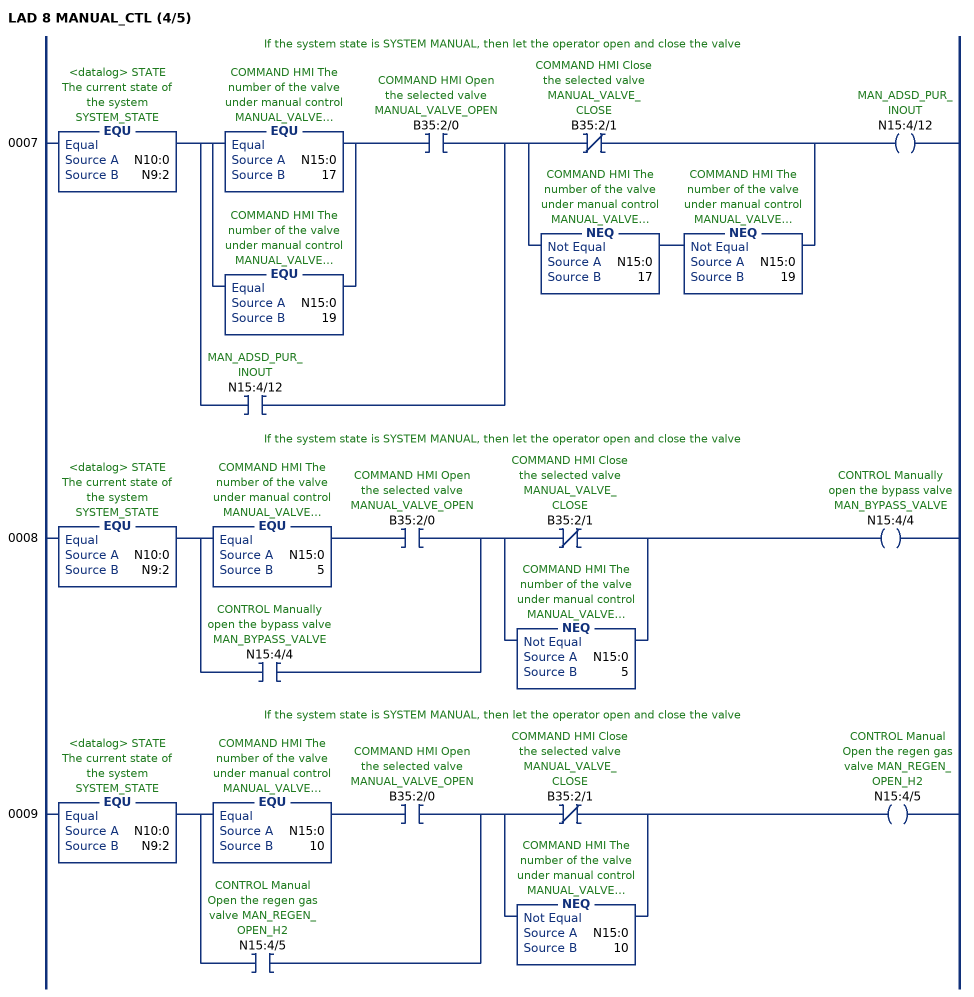
% Rung: 7 %
% If the system state is SYSTEM MANUAL, then let the operator open and close the valve %
SOR EQU N10:0 N9:2 BST BST EQU N15:0 17 NXB EQU N15:0 19 BND XIC B35:2/0 NXB XIC N15:4/12 BND BST XIO B35:2/1 NXB NEQ N15:0 17 NEQ N15:0 19 BND OTE N15:4/12 EOR
%   N10:0  SYSTEM_STATE  "<datalog> STATE The current state of the system" %
%   N9:2  SYSTEM_MANUAL  "STATE System Manual" %
%   N15:0  MANUAL_VALVE_NUMBER  "COMMAND HMI The number of the valve under manual control" %
%   B35:2/0  MANUAL_VALVE_OPEN  "COMMAND HMI Open the selected valve" %
%   N15:4/12  MAN_ADSD_PUR_INOUT %
%   B35:2/1  MANUAL_VALVE_CLOSE  "COMMAND HMI Close the selected valve" %
% Rung: 8 %
% If the system state is SYSTEM MANUAL, then let the operator open and close the valve %
SOR EQU N10:0 N9:2 BST EQU N15:0 5 XIC B35:2/0 NXB XIC N15:4/4 BND BST XIO B35:2/1 NXB NEQ N15:0 5 BND OTE N15:4/4 EOR
%   N10:0  SYSTEM_STATE  "<datalog> STATE The current state of the system" %
%   N9:2  SYSTEM_MANUAL  "STATE System Manual" %
%   N15:0  MANUAL_VALVE_NUMBER  "COMMAND HMI The number of the valve under manual control" %
%   B35:2/0  MANUAL_VALVE_OPEN  "COMMAND HMI Open the selected valve" %
%   N15:4/4  MAN_BYPASS_VALVE  "CONTROL Manually open the bypass valve" %
%   B35:2/1  MANUAL_VALVE_CLOSE  "COMMAND HMI Close the selected valve" %
% Rung: 9 %
% If the system state is SYSTEM MANUAL, then let the operator open and close the valve %
SOR EQU N10:0 N9:2 BST EQU N15:0 10 XIC B35:2/0 NXB XIC N15:4/5 BND BST XIO B35:2/1 NXB NEQ N15:0 10 BND OTE N15:4/5 EOR
%   N10:0  SYSTEM_STATE  "<datalog> STATE The current state of the system" %
%   N9:2  SYSTEM_MANUAL  "STATE System Manual" %
%   N15:0  MANUAL_VALVE_NUMBER  "COMMAND HMI The number of the valve under manual control" %
%   B35:2/0  MANUAL_VALVE_OPEN  "COMMAND HMI Open the selected valve" %
%   N15:4/5  MAN_REGEN_OPEN_H2  "CONTROL Manual Open the regen gas valve" %
%   B35:2/1  MANUAL_VALVE_CLOSE  "COMMAND HMI Close the selected valve" %

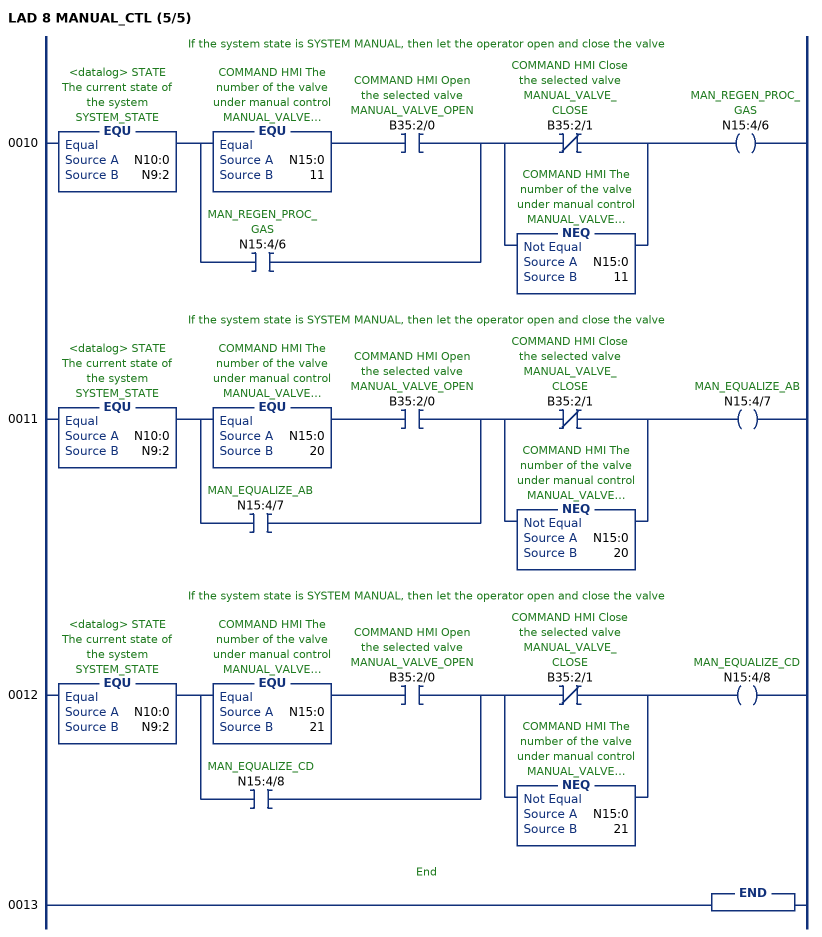
% Rung: 10 %
% If the system state is SYSTEM MANUAL, then let the operator open and close the valve %
SOR EQU N10:0 N9:2 BST EQU N15:0 11 XIC B35:2/0 NXB XIC N15:4/6 BND BST XIO B35:2/1 NXB NEQ N15:0 11 BND OTE N15:4/6 EOR
%   N10:0  SYSTEM_STATE  "<datalog> STATE The current state of the system" %
%   N9:2  SYSTEM_MANUAL  "STATE System Manual" %
%   N15:0  MANUAL_VALVE_NUMBER  "COMMAND HMI The number of the valve under manual control" %
%   B35:2/0  MANUAL_VALVE_OPEN  "COMMAND HMI Open the selected valve" %
%   N15:4/6  MAN_REGEN_PROC_GAS %
%   B35:2/1  MANUAL_VALVE_CLOSE  "COMMAND HMI Close the selected valve" %
% Rung: 11 %
% If the system state is SYSTEM MANUAL, then let the operator open and close the valve %
SOR EQU N10:0 N9:2 BST EQU N15:0 20 XIC B35:2/0 NXB XIC N15:4/7 BND BST XIO B35:2/1 NXB NEQ N15:0 20 BND OTE N15:4/7 EOR
%   N10:0  SYSTEM_STATE  "<datalog> STATE The current state of the system" %
%   N9:2  SYSTEM_MANUAL  "STATE System Manual" %
%   N15:0  MANUAL_VALVE_NUMBER  "COMMAND HMI The number of the valve under manual control" %
%   B35:2/0  MANUAL_VALVE_OPEN  "COMMAND HMI Open the selected valve" %
%   N15:4/7  MAN_EQUALIZE_AB %
%   B35:2/1  MANUAL_VALVE_CLOSE  "COMMAND HMI Close the selected valve" %
% Rung: 12 %
% If the system state is SYSTEM MANUAL, then let the operator open and close the valve %
SOR EQU N10:0 N9:2 BST EQU N15:0 21 XIC B35:2/0 NXB XIC N15:4/8 BND BST XIO B35:2/1 NXB NEQ N15:0 21 BND OTE N15:4/8 EOR
%   N10:0  SYSTEM_STATE  "<datalog> STATE The current state of the system" %
%   N9:2  SYSTEM_MANUAL  "STATE System Manual" %
%   N15:0  MANUAL_VALVE_NUMBER  "COMMAND HMI The number of the valve under manual control" %
%   B35:2/0  MANUAL_VALVE_OPEN  "COMMAND HMI Open the selected valve" %
%   N15:4/8  MAN_EQUALIZE_CD %
%   B35:2/1  MANUAL_VALVE_CLOSE  "COMMAND HMI Close the selected valve" %
% Rung: 13 %
% End %
SOR END EOR

LADDER 10 "PURIFY"    % Operates the purify control %
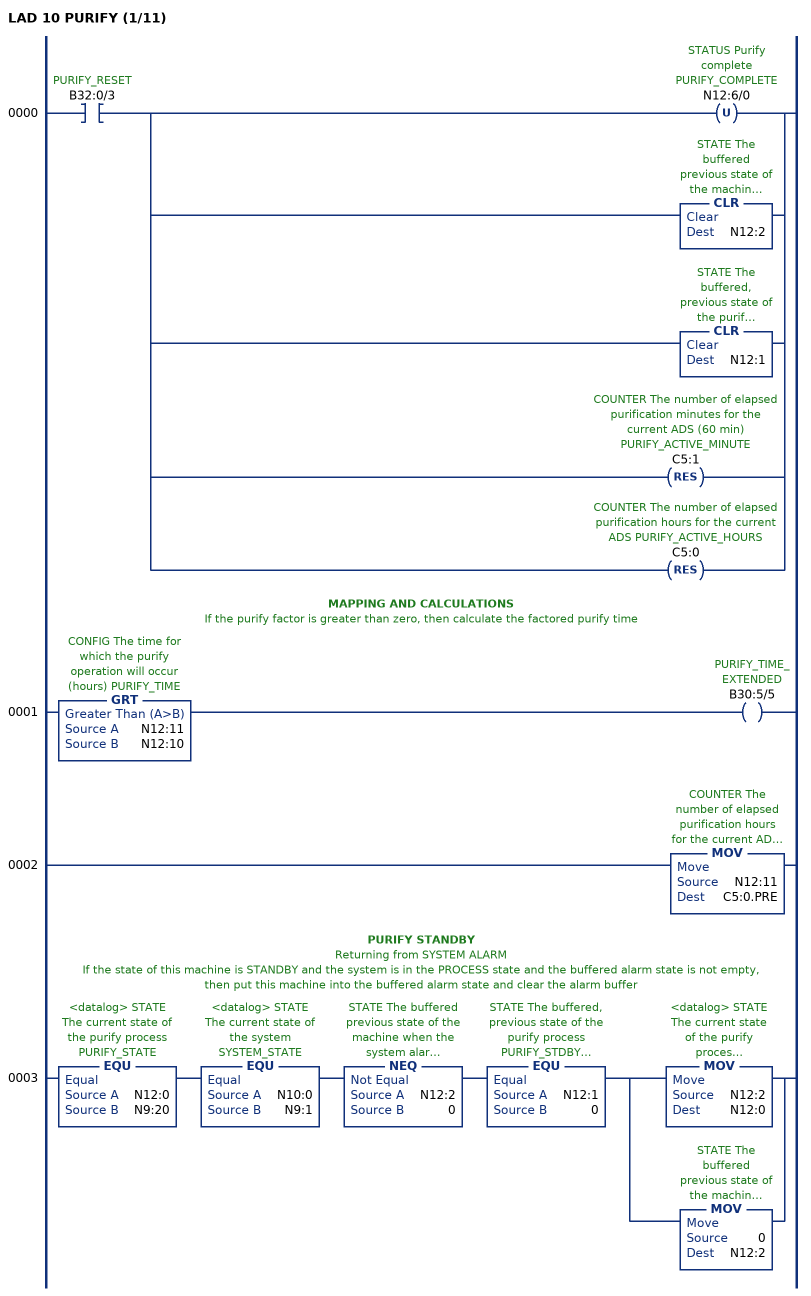
% Rung: 0 %
SOR XIC B32:0/3 BST OTU N12:6/0 NXB CLR N12:2 NXB CLR N12:1 NXB RES C5:1 NXB RES C5:0 BND EOR
%   B32:0/3  PURIFY_RESET %
%   N12:6/0  PURIFY_COMPLETE  "STATUS Purify complete" %
%   N12:2  PURIFY_ALARM_BUFFER  "STATE The buffered previous state of the machine when the system alarm occured" %
%   N12:1  PURIFY_STDBY_BUFFER  "STATE The buffered, previous state of the purify process" %
%   C5:1  PURIFY_ACTIVE_MINUTE  "COUNTER The number of elapsed purification minutes for the current ADS (60 min)" %
%   C5:0  PURIFY_ACTIVE_HOURS  "COUNTER The number of elapsed purification hours for the current ADS" %
% Rung: 1 %
% TITLE: MAPPING AND CALCULATIONS %
% If the purify factor is greater than zero, then calculate the factored purify time %
SOR GRT N12:11 N12:10 OTE B30:5/5 EOR
%   N12:11  PURIFY_TIME  "CONFIG The time for which the purify operation will occur (hours)" %
%   N12:10  DEFAULT_PURIFY_TIME  "CONFIG The percent output requested by the operator (percent)" %
%   B30:5/5  PURIFY_TIME_EXTENDED %
% Rung: 2 %
SOR MOV N12:11 C5:0.PRE EOR
%   N12:11  PURIFY_TIME  "CONFIG The time for which the purify operation will occur (hours)" %
%   C5:0  PURIFY_ACTIVE_HOURS  "COUNTER The number of elapsed purification hours for the current ADS" %
% Rung: 3 %
% TITLE: PURIFY STANDBY %
% Returning from SYSTEM ALARM
% If the state of this machine is STANDBY and the system is in the PROCESS state and the buffered alarm state is not empty, then put this machine into the buffered alarm state and clear the alarm buffer %
SOR EQU N12:0 N9:20 EQU N10:0 N9:1 NEQ N12:2 0 EQU N12:1 0 BST MOV N12:2 N12:0 NXB MOV 0 N12:2 BND EOR
%   N12:0  PURIFY_STATE  "<datalog> STATE The current state of the purify process" %
%   N9:20  PURIFY_STANDBY  "STATE Purify Standby" %
%   N10:0  SYSTEM_STATE  "<datalog> STATE The current state of the system" %
%   N9:1  SYSTEM_PROCESS  "STATE System Process" %
%   N12:2  PURIFY_ALARM_BUFFER  "STATE The buffered previous state of the machine when the system alarm occured" %
%   N12:1  PURIFY_STDBY_BUFFER  "STATE The buffered, previous state of the purify process" %

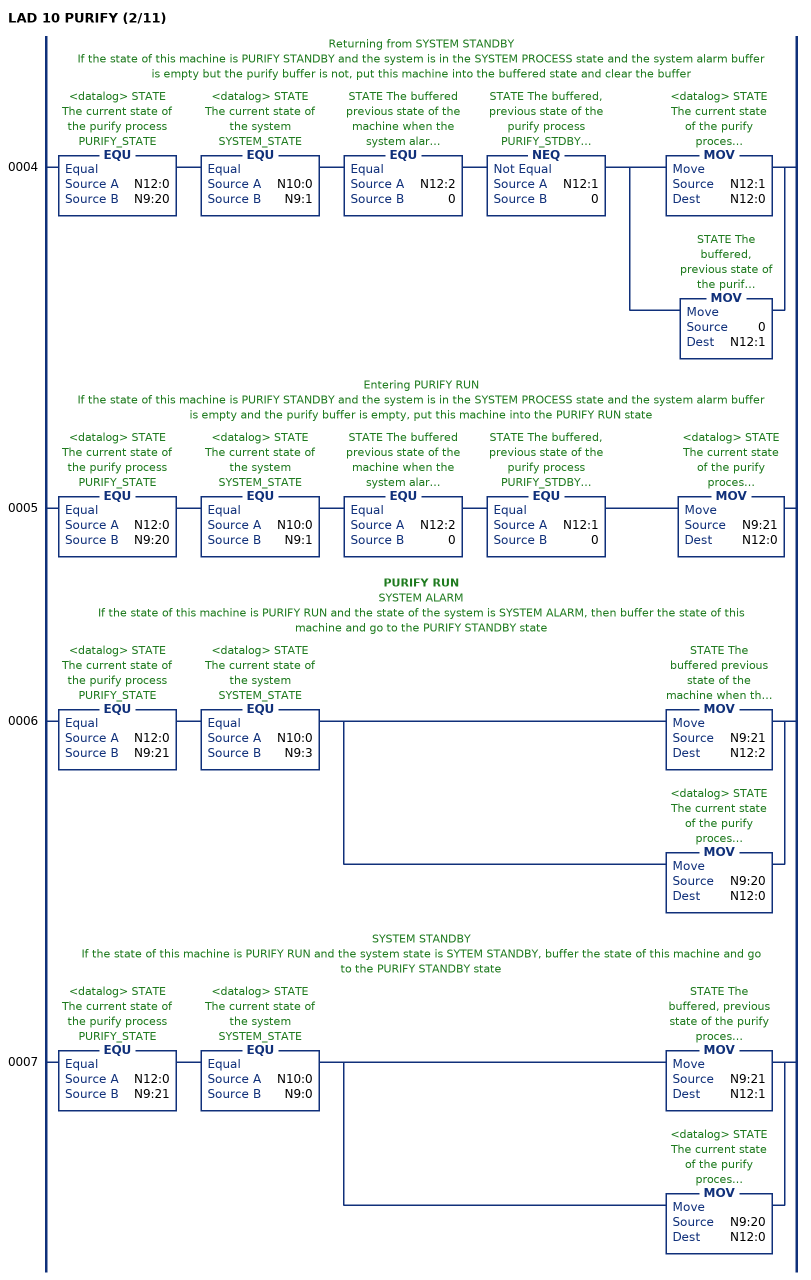
% Rung: 4 %
% Returning from SYSTEM STANDBY
% If the state of this machine is PURIFY STANDBY and the system is in the SYSTEM PROCESS state and the system alarm buffer is empty but the purify buffer is not, put this machine into the buffered state and clear the buffer %
SOR EQU N12:0 N9:20 EQU N10:0 N9:1 EQU N12:2 0 NEQ N12:1 0 BST MOV N12:1 N12:0 NXB MOV 0 N12:1 BND EOR
%   N12:0  PURIFY_STATE  "<datalog> STATE The current state of the purify process" %
%   N9:20  PURIFY_STANDBY  "STATE Purify Standby" %
%   N10:0  SYSTEM_STATE  "<datalog> STATE The current state of the system" %
%   N9:1  SYSTEM_PROCESS  "STATE System Process" %
%   N12:2  PURIFY_ALARM_BUFFER  "STATE The buffered previous state of the machine when the system alarm occured" %
%   N12:1  PURIFY_STDBY_BUFFER  "STATE The buffered, previous state of the purify process" %
% Rung: 5 %
% Entering PURIFY RUN
% If the state of this machine is PURIFY STANDBY and the system is in the SYSTEM PROCESS state and the system alarm buffer is empty and the purify buffer is empty, put this machine into the PURIFY RUN state %
SOR EQU N12:0 N9:20 EQU N10:0 N9:1 EQU N12:2 0 EQU N12:1 0 MOV N9:21 N12:0 EOR
%   N12:0  PURIFY_STATE  "<datalog> STATE The current state of the purify process" %
%   N9:20  PURIFY_STANDBY  "STATE Purify Standby" %
%   N10:0  SYSTEM_STATE  "<datalog> STATE The current state of the system" %
%   N9:1  SYSTEM_PROCESS  "STATE System Process" %
%   N12:2  PURIFY_ALARM_BUFFER  "STATE The buffered previous state of the machine when the system alarm occured" %
%   N12:1  PURIFY_STDBY_BUFFER  "STATE The buffered, previous state of the purify process" %
%   N9:21  PURIFY_RUN  "STATE Purify running" %
% Rung: 6 %
% TITLE: PURIFY RUN %
% SYSTEM ALARM
% If the state of this machine is PURIFY RUN and the state of the system is SYSTEM ALARM, then buffer the state of this machine and go to the PURIFY STANDBY state %
SOR EQU N12:0 N9:21 EQU N10:0 N9:3 BST MOV N9:21 N12:2 NXB MOV N9:20 N12:0 BND EOR
%   N12:0  PURIFY_STATE  "<datalog> STATE The current state of the purify process" %
%   N9:21  PURIFY_RUN  "STATE Purify running" %
%   N10:0  SYSTEM_STATE  "<datalog> STATE The current state of the system" %
%   N9:3  SYSTEM_ALARM  "STATE System Alarm" %
%   N12:2  PURIFY_ALARM_BUFFER  "STATE The buffered previous state of the machine when the system alarm occured" %
%   N9:20  PURIFY_STANDBY  "STATE Purify Standby" %
% Rung: 7 %
% SYSTEM STANDBY
% If the state of this machine is PURIFY RUN and the system state is SYTEM STANDBY, buffer the state of this machine and go to the PURIFY STANDBY state %
SOR EQU N12:0 N9:21 EQU N10:0 N9:0 BST MOV N9:21 N12:1 NXB MOV N9:20 N12:0 BND EOR
%   N12:0  PURIFY_STATE  "<datalog> STATE The current state of the purify process" %
%   N9:21  PURIFY_RUN  "STATE Purify running" %
%   N10:0  SYSTEM_STATE  "<datalog> STATE The current state of the system" %
%   N9:0  SYSTEM_STANDBY  "STATE System Standby" %
%   N12:1  PURIFY_STDBY_BUFFER  "STATE The buffered, previous state of the purify process" %
%   N9:20  PURIFY_STANDBY  "STATE Purify Standby" %

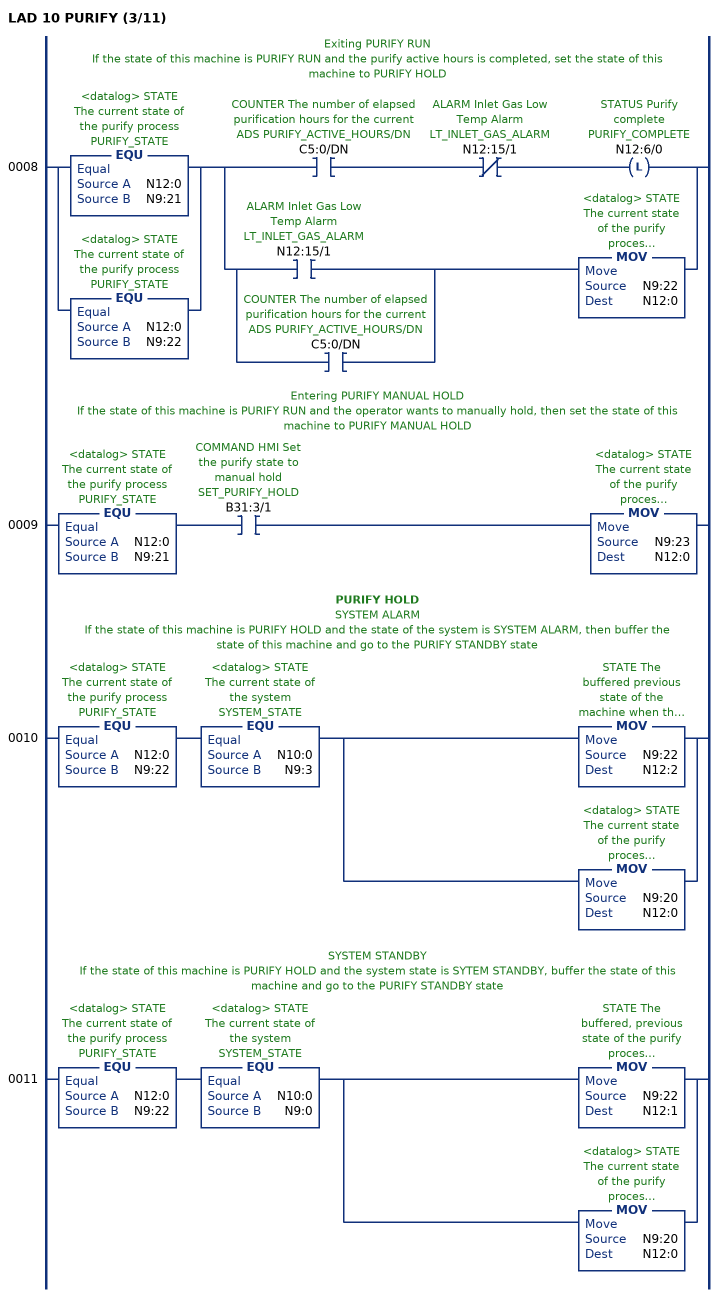
% Rung: 8 %
% Exiting PURIFY RUN
% If the state of this machine is PURIFY RUN and the purify active hours is completed, set the state of this machine to PURIFY HOLD %
SOR BST EQU N12:0 N9:21 NXB EQU N12:0 N9:22 BND BST XIC C5:0/DN XIO N12:15/1 OTL N12:6/0 NXB BST XIC N12:15/1 NXB XIC C5:0/DN BND MOV N9:22 N12:0 BND EOR
%   N12:0  PURIFY_STATE  "<datalog> STATE The current state of the purify process" %
%   N9:21  PURIFY_RUN  "STATE Purify running" %
%   N9:22  PURIFY_HOLD  "STATE Purify Hold" %
%   C5:0  PURIFY_ACTIVE_HOURS  "COUNTER The number of elapsed purification hours for the current ADS" %
%   N12:15/1  LT_INLET_GAS_ALARM  "ALARM Inlet Gas Low Temp Alarm" %
%   N12:6/0  PURIFY_COMPLETE  "STATUS Purify complete" %
% Rung: 9 %
% Entering PURIFY MANUAL HOLD
% If the state of this machine is PURIFY RUN and the operator wants to manually hold, then set the state of this machine to PURIFY MANUAL HOLD %
SOR EQU N12:0 N9:21 XIC B31:3/1 MOV N9:23 N12:0 EOR
%   N12:0  PURIFY_STATE  "<datalog> STATE The current state of the purify process" %
%   N9:21  PURIFY_RUN  "STATE Purify running" %
%   B31:3/1  SET_PURIFY_HOLD  "COMMAND HMI Set the purify state to manual hold" %
%   N9:23  PURIFY_MANUAL_HOLD  "STATE Purify Manual Hold" %
% Rung: 10 %
% TITLE: PURIFY HOLD %
% SYSTEM ALARM
% If the state of this machine is PURIFY HOLD and the state of the system is SYSTEM ALARM, then buffer the state of this machine and go to the PURIFY STANDBY state %
SOR EQU N12:0 N9:22 EQU N10:0 N9:3 BST MOV N9:22 N12:2 NXB MOV N9:20 N12:0 BND EOR
%   N12:0  PURIFY_STATE  "<datalog> STATE The current state of the purify process" %
%   N9:22  PURIFY_HOLD  "STATE Purify Hold" %
%   N10:0  SYSTEM_STATE  "<datalog> STATE The current state of the system" %
%   N9:3  SYSTEM_ALARM  "STATE System Alarm" %
%   N12:2  PURIFY_ALARM_BUFFER  "STATE The buffered previous state of the machine when the system alarm occured" %
%   N9:20  PURIFY_STANDBY  "STATE Purify Standby" %
% Rung: 11 %
% SYSTEM STANDBY
% If the state of this machine is PURIFY HOLD and the system state is SYTEM STANDBY, buffer the state of this machine and go to the PURIFY STANDBY state %
SOR EQU N12:0 N9:22 EQU N10:0 N9:0 BST MOV N9:22 N12:1 NXB MOV N9:20 N12:0 BND EOR
%   N12:0  PURIFY_STATE  "<datalog> STATE The current state of the purify process" %
%   N9:22  PURIFY_HOLD  "STATE Purify Hold" %
%   N10:0  SYSTEM_STATE  "<datalog> STATE The current state of the system" %
%   N9:0  SYSTEM_STANDBY  "STATE System Standby" %
%   N12:1  PURIFY_STDBY_BUFFER  "STATE The buffered, previous state of the purify process" %
%   N9:20  PURIFY_STANDBY  "STATE Purify Standby" %

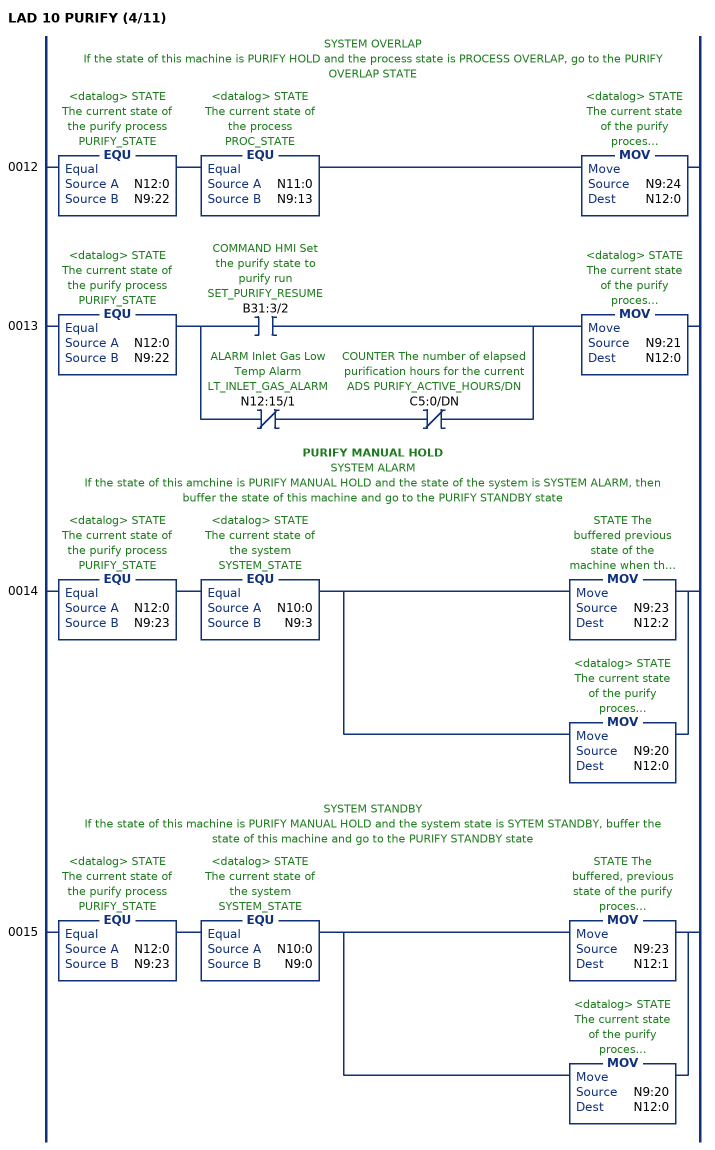
% Rung: 12 %
% SYSTEM OVERLAP
% If the state of this machine is PURIFY HOLD and the process state is PROCESS OVERLAP, go to the PURIFY OVERLAP STATE %
SOR EQU N12:0 N9:22 EQU N11:0 N9:13 MOV N9:24 N12:0 EOR
%   N12:0  PURIFY_STATE  "<datalog> STATE The current state of the purify process" %
%   N9:22  PURIFY_HOLD  "STATE Purify Hold" %
%   N11:0  PROC_STATE  "<datalog> STATE The current state of the process" %
%   N9:13  PROC_OVERLAP  "STATE Process Purify Overlap" %
%   N9:24  PURIFY_OVERLAP  "STATE Puriify Overlap" %
% Rung: 13 %
SOR EQU N12:0 N9:22 BST XIC B31:3/2 NXB XIO N12:15/1 XIO C5:0/DN BND MOV N9:21 N12:0 EOR
%   N12:0  PURIFY_STATE  "<datalog> STATE The current state of the purify process" %
%   N9:22  PURIFY_HOLD  "STATE Purify Hold" %
%   B31:3/2  SET_PURIFY_RESUME  "COMMAND HMI Set the purify state to purify run" %
%   N12:15/1  LT_INLET_GAS_ALARM  "ALARM Inlet Gas Low Temp Alarm" %
%   C5:0  PURIFY_ACTIVE_HOURS  "COUNTER The number of elapsed purification hours for the current ADS" %
%   N9:21  PURIFY_RUN  "STATE Purify running" %
% Rung: 14 %
% TITLE: PURIFY MANUAL HOLD %
% SYSTEM ALARM
% If the state of this amchine is PURIFY MANUAL HOLD and the state of the system is SYSTEM ALARM, then buffer the state of this machine and go to the PURIFY STANDBY state %
SOR EQU N12:0 N9:23 EQU N10:0 N9:3 BST MOV N9:23 N12:2 NXB MOV N9:20 N12:0 BND EOR
%   N12:0  PURIFY_STATE  "<datalog> STATE The current state of the purify process" %
%   N9:23  PURIFY_MANUAL_HOLD  "STATE Purify Manual Hold" %
%   N10:0  SYSTEM_STATE  "<datalog> STATE The current state of the system" %
%   N9:3  SYSTEM_ALARM  "STATE System Alarm" %
%   N12:2  PURIFY_ALARM_BUFFER  "STATE The buffered previous state of the machine when the system alarm occured" %
%   N9:20  PURIFY_STANDBY  "STATE Purify Standby" %
% Rung: 15 %
% SYSTEM STANDBY
% If the state of this machine is PURIFY MANUAL HOLD and the system state is SYTEM STANDBY, buffer the state of this machine and go to the PURIFY STANDBY state %
SOR EQU N12:0 N9:23 EQU N10:0 N9:0 BST MOV N9:23 N12:1 NXB MOV N9:20 N12:0 BND EOR
%   N12:0  PURIFY_STATE  "<datalog> STATE The current state of the purify process" %
%   N9:23  PURIFY_MANUAL_HOLD  "STATE Purify Manual Hold" %
%   N10:0  SYSTEM_STATE  "<datalog> STATE The current state of the system" %
%   N9:0  SYSTEM_STANDBY  "STATE System Standby" %
%   N12:1  PURIFY_STDBY_BUFFER  "STATE The buffered, previous state of the purify process" %
%   N9:20  PURIFY_STANDBY  "STATE Purify Standby" %

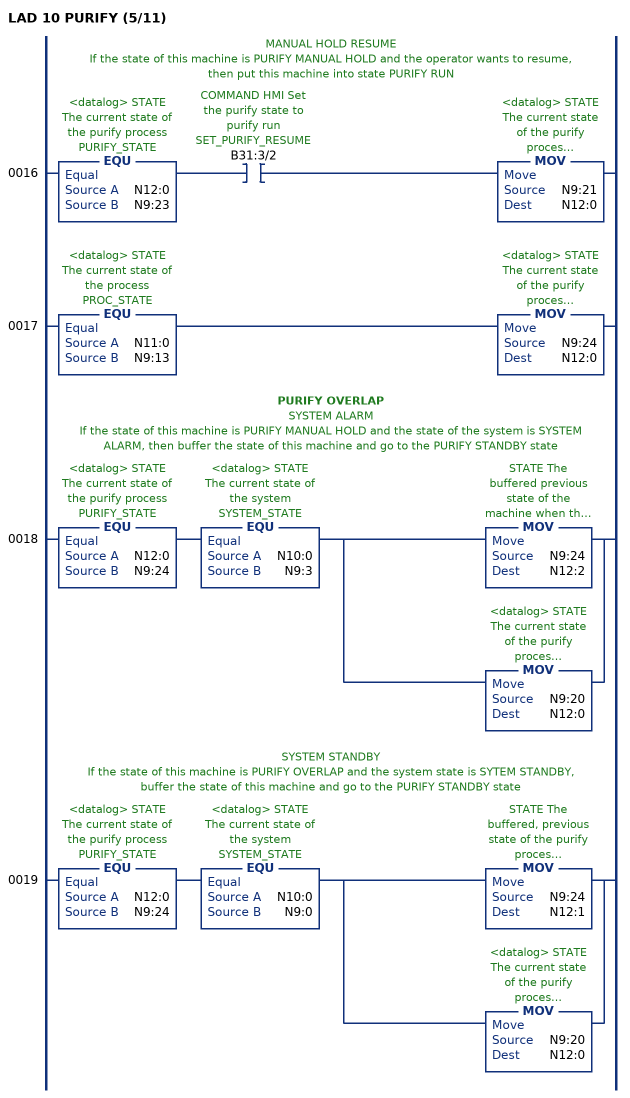
% Rung: 16 %
% MANUAL HOLD RESUME
% If the state of this machine is PURIFY MANUAL HOLD and the operator wants to resume, then put this machine into state PURIFY RUN %
SOR EQU N12:0 N9:23 XIC B31:3/2 MOV N9:21 N12:0 EOR
%   N12:0  PURIFY_STATE  "<datalog> STATE The current state of the purify process" %
%   N9:23  PURIFY_MANUAL_HOLD  "STATE Purify Manual Hold" %
%   B31:3/2  SET_PURIFY_RESUME  "COMMAND HMI Set the purify state to purify run" %
%   N9:21  PURIFY_RUN  "STATE Purify running" %
% Rung: 17 %
SOR EQU N11:0 N9:13 MOV N9:24 N12:0 EOR
%   N11:0  PROC_STATE  "<datalog> STATE The current state of the process" %
%   N9:13  PROC_OVERLAP  "STATE Process Purify Overlap" %
%   N9:24  PURIFY_OVERLAP  "STATE Puriify Overlap" %
%   N12:0  PURIFY_STATE  "<datalog> STATE The current state of the purify process" %
% Rung: 18 %
% TITLE: PURIFY OVERLAP %
% SYSTEM ALARM
% If the state of this machine is PURIFY MANUAL HOLD and the state of the system is SYSTEM ALARM, then buffer the state of this machine and go to the PURIFY STANDBY state %
SOR EQU N12:0 N9:24 EQU N10:0 N9:3 BST MOV N9:24 N12:2 NXB MOV N9:20 N12:0 BND EOR
%   N12:0  PURIFY_STATE  "<datalog> STATE The current state of the purify process" %
%   N9:24  PURIFY_OVERLAP  "STATE Puriify Overlap" %
%   N10:0  SYSTEM_STATE  "<datalog> STATE The current state of the system" %
%   N9:3  SYSTEM_ALARM  "STATE System Alarm" %
%   N12:2  PURIFY_ALARM_BUFFER  "STATE The buffered previous state of the machine when the system alarm occured" %
%   N9:20  PURIFY_STANDBY  "STATE Purify Standby" %
% Rung: 19 %
% SYSTEM STANDBY
% If the state of this machine is PURIFY OVERLAP and the system state is SYTEM STANDBY, buffer the state of this machine and go to the PURIFY STANDBY state %
SOR EQU N12:0 N9:24 EQU N10:0 N9:0 BST MOV N9:24 N12:1 NXB MOV N9:20 N12:0 BND EOR
%   N12:0  PURIFY_STATE  "<datalog> STATE The current state of the purify process" %
%   N9:24  PURIFY_OVERLAP  "STATE Puriify Overlap" %
%   N10:0  SYSTEM_STATE  "<datalog> STATE The current state of the system" %
%   N9:0  SYSTEM_STANDBY  "STATE System Standby" %
%   N12:1  PURIFY_STDBY_BUFFER  "STATE The buffered, previous state of the purify process" %
%   N9:20  PURIFY_STANDBY  "STATE Purify Standby" %

